// TIA Portal project "cpsforge_tiaportal" (V17)

(* hardware
DEVICE "S7-1200 station_1"  S7-1200 Station
   slot 0: "Rack_0"  S7-1200 Rack  Rack  V1.0
   slot 1: "PLC_1"  CPU 1212FC DC/DC/RLY  6ES7 212-1HF40-0XB0  V4.5
*)

// ===== PLC "PLC_1"  CPU 1212FC DC/DC/RLY =====

VAR_GLOBAL   // PLC tag table "Default tag table"
   "Tag__639094376035440745" AT %I0.0 : Bool;
   "Tag__639094376037924724" AT %Q0.0 : Bool;
   "Tag__639094376037924725" AT %I0.1 : Bool;
   "Tag__639094376038085904" AT %Q0.1 : Bool;
   "Tag__639094376038085905" AT %Q0.2 : Bool;
   "Tag__639094376038245632" AT %I0.2 : Bool;
   "Tag__639094376038245633" AT %I0.3 : Bool;
   "Tag__639094376038405651" AT %I0.4 : Bool;
   "Tag__639094376038405652" AT %I0.5 : Bool;
   "Tag__639094376038405653" AT %Q0.3 : Bool;
   "Tag__639094376038565707" AT %Q0.4 : Bool;
   "Tag__639094376038565708" AT %Q0.5 : Bool;
   "Tag__639094376038565709" AT %Q1.0 : Bool;
   "Tag__639094376038885860" AT %I10.0 : Bool;
   "Tag__639094376038885861" AT %I10.1 : Bool;
   "Tag__639094376039046363" AT %I10.2 : Bool;
   "Tag__639094376039046364" AT %I10.3 : Bool;
   "Tag__639094376039046365" AT %I10.4 : Bool;
   "Tag__639094376039205258" AT %I10.5 : Bool;
   "Tag__639094376039205259" AT %I10.6 : Bool;
   "Tag__639094376039205260" AT %I10.7 : Bool;
   "Tag__639094376039365268" AT %I11.0 : Bool;
   "Tag__639094376039365269" AT %I11.1 : Bool;
   "Tag__639094376039365270" AT %I11.2 : Bool;
   "Tag__639094376039525211" AT %I11.3 : Bool;
   "Tag__639094376039525212" AT %I11.4 : Bool;
   "Tag__639094376039525213" AT %I11.5 : Bool;
   "Tag__639094376039685481" AT %I11.6 : Bool;
   "Tag__639094376039685482" AT %I11.7 : Bool;
   "Tag__639094376039685483" AT %I12.0 : Bool;
   "Tag__639094376039846408" AT %I12.1 : Bool;
   "Tag__639094376039846409" AT %I12.2 : Bool;
   "Tag__639094376039846410" AT %Q0.6 : Bool;
   "Tag__639094376040005546" AT %Q0.7 : Bool;
   "Tag__639094376040005547" AT %Q1.1 : Bool;
   "Tag__639094376040005548" AT %Q1.2 : Bool;
   "Tag__639094376040163908" AT %Q1.3 : Bool;
   "Tag__639094376040163909" AT %Q1.4 : Bool;
   "Tag__639094376040163910" AT %Q1.5 : Bool;
   "Tag__639094376040323143" AT %Q1.6 : Bool;
   "Tag__639094376040323144" AT %Q1.7 : Bool;
   "Tag__639094376040323145" AT %Q2.0 : Bool;
   "Tag__639094376040483081" AT %Q2.1 : Bool;
   "Tag__639094376040483082" AT %Q2.2 : Bool;
   "Tag__639094376040483083" AT %Q2.3 : Bool;
   "Tag__639094376040642647" AT %Q2.4 : Bool;
   "Tag__639094376040642648" AT %Q2.5 : Bool;
   "Tag__639094376040642649" AT %Q2.6 : Bool;
   "Tag__639094376040802767" AT %Q2.7 : Bool;
   "Tag__639094376040802768" AT %Q3.0 : Bool;
   "Tag__639094376040802769" AT %Q3.1 : Bool;
   "Tag__639094376040963045" AT %QD100 : DWord;
   "Tag__639094376041124518" AT %I12.3 : Bool;
   "Tag__639094376041124519" AT %I12.4 : Bool;
   "Tag__639094376041283188" AT %I12.5 : Bool;
   "Tag__639094376041283189" AT %I12.6 : Bool;
   "Tag__639094376041283190" AT %I12.7 : Bool;
   "Tag__639094376041442043" AT %I13.0 : Bool;
   "Tag__639094376041442044" AT %I13.1 : Bool;
   "Tag__639094376041600752" AT %I13.2 : Bool;
   "Tag__639094376041600753" AT %I13.3 : Bool;
   "Tag__639094376041600754" AT %I13.4 : Bool;
   "Tag__639094376041760860" AT %Q3.2 : Bool;
   "Tag__639094376041918319" AT %Q3.3 : Bool;
   "Tag__639094376041918320" AT %Q3.4 : Bool;
   "Tag__639094376042076147" AT %ID100 : DWord;
   "Tag__639094376042076148" AT %ID104 : DWord;
   "Tag__639094376042235578" AT %ID108 : DWord;
   "Tag__639094376042315926" AT %QD104 : DWord;
   "Tag__639094376042397245" AT %QD108 : DWord;
   "Tag__639094376042397246" AT %QD112 : DWord;
   "Tag__639094376042713202" AT %I0.6 : Bool;
   "Tag__639094376042871627" AT %I0.7 : Bool;
   "Tag__639094376042871628" AT %I1.0 : Bool;
   "Tag__639094376043030339" AT %I1.1 : Bool;
   "Tag__639094376043070322" AT %I1.2 : Bool;
   "Tag__639094376043147186" AT %I1.3 : Bool;
   "Tag__639094376043188096" AT %I1.4 : Bool;
   "Tag__639094376043188097" AT %I1.5 : Bool;
   "Tag__639094376043188098" AT %I1.6 : Bool;
   "Tag__639094376043345950" AT %I1.7 : Bool;
   "Tag__639094559022291825" AT %QB0 : Byte;
   "Tag__639094559022387271" AT %QB1 : Byte;
   "Tag__639094559022442425" AT %QB2 : Byte;
   "Tag__639094559022502581" AT %QB3 : Byte;
END_VAR

DATA_BLOCK "DB_Config"   // DB2
{ S7_Optimized_Access := 'FALSE' }
VERSION : 0.1
// MANTIS â€” DB_Config: Global configuration block
//  ActiveScene selects which Factory I/O scene is running
   VAR
      ActiveScene : Int := 19;   // Default: Sorting Height Basic
      ScanRate_ms : Int := 1000;   // Control loop period
      Running : Bool := TRUE;   // System running flag
   END_VAR
BEGIN
END_DATA_BLOCK

DATA_BLOCK "FB_FromAtoB_DB"   // DB3
{ S7_Optimized_Access := 'FALSE' }
VERSION : 0.1
// =============================================================================
//  MANTIS â€” Instance Data Blocks for all 21 Factory I/O Scene FBs
// 
//  After importing this file in TIA Portal, you MUST set the DB numbers:
//    Right-click each DB â†’ Properties â†’ General â†’ Number
//    Assign the DB numbers according to the table below.
// 
//  DB Number Assignments:
//    DB10 = FB_FromAtoB_DB
//    DB11 = FB_FromAtoB_SR_DB
//    DB12 = FB_FillingTank_DB
//    DB13 = FB_QueueItems_DB
//    DB14 = FB_Assembler_DB
//    DB15 = FB_AssemblerAnalog_DB
//    DB16 = FB_Warehouse_DB
//    DB17 = FB_BufferStation_DB
//    DB18 = FB_ConvergeStation_DB
//    DB19 = FB_ElevatorAdvanced_DB
//    DB20 = FB_ElevatorBasic_DB
//    DB21 = FB_LevelControl_DB
//    DB22 = FB_Palletizer_DB
//    DB23 = FB_PickPlaceBasic_DB
//    DB24 = FB_PickPlaceXYZ_DB
//    DB25 = FB_ProductionLine_DB
//    DB26 = FB_SeparatingStation_DB
//    DB27 = FB_SortingHeightAdv_DB
//    DB28 = FB_SortingHeightBasic_DB
//    DB29 = FB_SortingWeight_DB
//    DB30 = FB_SortingStation_DB
//  =============================================================================
//  Scene 1: From A to B â†’ DB10
// stored: InstanceOfName FB_FromAtoB
"FB_FromAtoB"
BEGIN
END_DATA_BLOCK

DATA_BLOCK "FB_FromAtoB_SR_DB"   // DB4
{ S7_Optimized_Access := 'FALSE' }
VERSION : 0.1
// Scene 2: From A to B (Set/Reset) â†’ DB11
// stored: InstanceOfName FB_FromAtoB_SR
"FB_FromAtoB_SR"
BEGIN
END_DATA_BLOCK

DATA_BLOCK "FB_FillingTank_DB"   // DB5
{ S7_Optimized_Access := 'FALSE' }
VERSION : 0.1
// Scene 3: Filling Tank â†’ DB12
// stored: InstanceOfName FB_FillingTank
"FB_FillingTank"
BEGIN
END_DATA_BLOCK

DATA_BLOCK "FB_QueueItems_DB"   // DB6
{ S7_Optimized_Access := 'FALSE' }
VERSION : 0.1
// Scene 4: Queue of Items â†’ DB13
// stored: InstanceOfName FB_QueueItems
"FB_QueueItems"
BEGIN
END_DATA_BLOCK

DATA_BLOCK "FB_Assembler_DB"   // DB7
{ S7_Optimized_Access := 'FALSE' }
VERSION : 0.1
// Scene 5: Assembler â†’ DB14
// stored: InstanceOfName FB_Assembler
"FB_Assembler"
BEGIN
END_DATA_BLOCK

DATA_BLOCK "FB_AssemblerAnalog_DB"   // DB8
{ S7_Optimized_Access := 'FALSE' }
VERSION : 0.1
// Scene 6: Assembler (Analog) â†’ DB15
// stored: InstanceOfName FB_AssemblerAnalog
"FB_AssemblerAnalog"
BEGIN
END_DATA_BLOCK

DATA_BLOCK "FB_Warehouse_DB"   // DB9
{ S7_Optimized_Access := 'FALSE' }
VERSION : 0.1
// Scene 7: Automated Warehouse â†’ DB16
// stored: InstanceOfName FB_Warehouse
"FB_Warehouse"
BEGIN
END_DATA_BLOCK

DATA_BLOCK "FB_BufferStation_DB"   // DB10
{ S7_Optimized_Access := 'FALSE' }
VERSION : 0.1
// Scene 8: Buffer Station â†’ DB17
// stored: InstanceOfName FB_BufferStation
"FB_BufferStation"
BEGIN
END_DATA_BLOCK

DATA_BLOCK "FB_ConvergeStation_DB"   // DB11
{ S7_Optimized_Access := 'FALSE' }
VERSION : 0.1
// Scene 9: Converge Station â†’ DB18
// stored: InstanceOfName FB_ConvergeStation
"FB_ConvergeStation"
BEGIN
END_DATA_BLOCK

DATA_BLOCK "FB_ElevatorAdvanced_DB"   // DB12
{ S7_Optimized_Access := 'FALSE' }
VERSION : 0.1
// Scene 10: Elevator (Advanced) â†’ DB19
// stored: InstanceOfName FB_ElevatorAdvanced
"FB_ElevatorAdvanced"
BEGIN
END_DATA_BLOCK

DATA_BLOCK "FB_ElevatorBasic_DB"   // DB13
{ S7_Optimized_Access := 'FALSE' }
VERSION : 0.1
// Scene 11: Elevator (Basic) â†’ DB20
// stored: InstanceOfName FB_ElevatorBasic
"FB_ElevatorBasic"
BEGIN
END_DATA_BLOCK

DATA_BLOCK "FB_LevelControl_DB"   // DB14
{ S7_Optimized_Access := 'FALSE' }
VERSION : 0.1
// Scene 12: Level Control â†’ DB21
// stored: InstanceOfName FB_LevelControl
"FB_LevelControl"
BEGIN
END_DATA_BLOCK

DATA_BLOCK "FB_Palletizer_DB"   // DB15
{ S7_Optimized_Access := 'FALSE' }
VERSION : 0.1
// Scene 13: Palletizer â†’ DB22
// stored: InstanceOfName FB_Palletizer
"FB_Palletizer"
BEGIN
END_DATA_BLOCK

DATA_BLOCK "FB_PickPlaceBasic_DB"   // DB16
{ S7_Optimized_Access := 'FALSE' }
VERSION : 0.1
// Scene 14: Pick & Place (Basic) â†’ DB23
// stored: InstanceOfName FB_PickPlaceBasic
"FB_PickPlaceBasic"
BEGIN
END_DATA_BLOCK

DATA_BLOCK "FB_PickPlaceXYZ_DB"   // DB17
{ S7_Optimized_Access := 'FALSE' }
VERSION : 0.1
// Scene 15: Pick & Place XYZ â†’ DB24
// stored: InstanceOfName FB_PickPlaceXYZ
"FB_PickPlaceXYZ"
BEGIN
END_DATA_BLOCK

DATA_BLOCK "FB_ProductionLine_DB"   // DB18
{ S7_Optimized_Access := 'FALSE' }
VERSION : 0.1
// Scene 16: Production Line â†’ DB25
// stored: InstanceOfName FB_ProductionLine
"FB_ProductionLine"
BEGIN
END_DATA_BLOCK

DATA_BLOCK "FB_SeparatingStation_DB"   // DB19
{ S7_Optimized_Access := 'FALSE' }
VERSION : 0.1
// Scene 17: Separating Station â†’ DB26
// stored: InstanceOfName FB_SeparatingStation
"FB_SeparatingStation"
BEGIN
END_DATA_BLOCK

DATA_BLOCK "FB_SortingHeightAdv_DB"   // DB20
{ S7_Optimized_Access := 'FALSE' }
VERSION : 0.1
// Scene 18: Sorting by Height (Advanced) â†’ DB27
// stored: InstanceOfName FB_SortingHeightAdvanced
"FB_SortingHeightAdvanced"
BEGIN
END_DATA_BLOCK

DATA_BLOCK "FB_SortingHeightBasic_DB"   // DB21
{ S7_Optimized_Access := 'FALSE' }
VERSION : 0.1
// Scene 19: Sorting by Height (Basic) â†’ DB28
// stored: InstanceOfName FB_SortingHeightBasic
"FB_SortingHeightBasic"
BEGIN
END_DATA_BLOCK

DATA_BLOCK "FB_SortingWeight_DB"   // DB22
{ S7_Optimized_Access := 'FALSE' }
VERSION : 0.1
// Scene 20: Sorting by Weight â†’ DB29
// stored: InstanceOfName FB_SortingWeight
"FB_SortingWeight"
BEGIN
END_DATA_BLOCK

DATA_BLOCK "FB_SortingStation_DB"   // DB23
{ S7_Optimized_Access := 'FALSE' }
VERSION : 0.1
// Scene 21: Sorting Station â†’ DB30
// stored: InstanceOfName FB_SortingStation
"FB_SortingStation"
BEGIN
END_DATA_BLOCK

FUNCTION_BLOCK "FB_Assembler"   // FB2, SCL
{ S7_Optimized_Access := 'FALSE' }
VERSION : 0.1
// MANTIS â€” Scene 5: Assembler
//  Assemble parts (lids + bases) using a two-axis pick and place.
//  DB14: I/O mapping
   VAR
      PartAtPickup : Bool;   // 0.0
      _pad0 : Byte;
      PartAtPlace : Bool;   // 2.0
      _pad1 : Byte;
      LidAtPickup : Bool;   // 4.0
      _pad2 : Byte;
      ClampSensor : Bool;   // 6.0
      _pad3 : Byte;
      MovingX : Bool;   // 8.0
      _pad4 : Byte;
      MovingZ : Bool;   // 10.0
      _pad5 : Byte;
      ConveyorBase : Bool;   // 12.0
      _pad6 : Byte;
      ConveyorLid : Bool;   // 14.0
      _pad7 : Byte;
      ConveyorOut : Bool;   // 16.0
      _pad8 : Byte;
      MoveX : Bool;   // 18.0
      _pad9 : Byte;
      MoveZ : Bool;   // 20.0
      _pad10 : Byte;
      Clamp : Bool;   // 22.0
      _pad11 : Byte;
      Emitter : Bool;   // 24.0
      _pad12 : Byte;
      iState : Int := 0;
   END_VAR
BEGIN
       CASE #iState OF
           0: // Feed base part
               #ConveyorBase := TRUE;
               #ConveyorLid := TRUE;
               #Emitter := TRUE;
               IF #PartAtPickup THEN
                   #ConveyorBase := FALSE;
                   #iState := 1;
               END_IF;

           1: // Move pick-and-place to pickup position
               #MoveX := FALSE;  // Move to pickup (left)
               #MoveZ := TRUE;   // Lower
               IF NOT #MovingZ THEN
                   #iState := 2;
               END_IF;

           2: // Clamp the part
               #Clamp := TRUE;
               IF #ClampSensor THEN
                   #MoveZ := FALSE;  // Raise
                   #iState := 3;
               END_IF;

           3: // Move to place position
               IF NOT #MovingZ THEN
                   #MoveX := TRUE;   // Move to place (right)
                   #iState := 4;
               END_IF;

           4: // Lower and place
               IF NOT #MovingX THEN
                   #MoveZ := TRUE;   // Lower
                   #iState := 5;
               END_IF;

           5: // Release
               IF NOT #MovingZ THEN
                   #Clamp := FALSE;
                   #MoveZ := FALSE;
                   #iState := 6;
               END_IF;

           6: // Output assembled part
               #ConveyorOut := TRUE;
               #MoveX := FALSE;  // Return to home
               IF NOT #PartAtPlace THEN
                   #ConveyorOut := FALSE;
                   #iState := 0;
               END_IF;
       END_CASE;
END_FUNCTION_BLOCK

FUNCTION_BLOCK "FB_AssemblerAnalog"   // FB3, SCL
{ S7_Optimized_Access := 'FALSE' }
VERSION : 0.1
// MANTIS â€” Scene 6: Assembler (Analog)
//  Assemble with analog position control for X/Z axes.
//  DB15: I/O mapping
   VAR
      PartAtPickup : Bool;   // 0.0
      _pad0 : Byte;
      PartAtPlace : Bool;   // 2.0
      _pad1 : Byte;
      LidAtPickup : Bool;   // 4.0
      _pad2 : Byte;
      ClampSensor : Bool;   // 6.0
      _pad3 : Byte;
      PosX : Real;   // 8
      PosZ : Real;   // 12
      ConveyorBase : Bool;   // 16.0
      _pad4 : Byte;
      ConveyorLid : Bool;   // 18.0
      _pad5 : Byte;
      ConveyorOut : Bool;   // 20.0
      _pad6 : Byte;
      SetpointX : Real;   // 22
      SetpointZ : Real;   // 26
      Clamp : Bool;   // 30.0
      _pad7 : Byte;
      Emitter : Bool;   // 32.0
      _pad8 : Byte;
      iState : Int := 0;
      PICKUP_X : Real := 100.0;
      PICKUP_Z : Real := 400.0;
      PLACE_X : Real := 800.0;
      PLACE_Z : Real := 400.0;
      HOME_Z : Real := 50.0;
      TOLERANCE : Real := 10.0;
   END_VAR
BEGIN
       CASE #iState OF
           0: // Feed parts
               #ConveyorBase := TRUE;
               #ConveyorLid := TRUE;
               #Emitter := TRUE;
               #SetpointX := #PICKUP_X;
               #SetpointZ := #HOME_Z;
               IF #PartAtPickup THEN
                   #ConveyorBase := FALSE;
                   #iState := 1;
               END_IF;

           1: // Move to pickup and lower
               #SetpointX := #PICKUP_X;
               #SetpointZ := #PICKUP_Z;
               IF ABS(#PosX - #PICKUP_X) < #TOLERANCE AND ABS(#PosZ - #PICKUP_Z) < #TOLERANCE THEN
                   #iState := 2;
               END_IF;

           2: // Clamp
               #Clamp := TRUE;
               IF #ClampSensor THEN
                   #SetpointZ := #HOME_Z;
                   #iState := 3;
               END_IF;

           3: // Raise and move to place
               IF ABS(#PosZ - #HOME_Z) < #TOLERANCE THEN
                   #SetpointX := #PLACE_X;
                   #iState := 4;
               END_IF;

           4: // Lower to place
               IF ABS(#PosX - #PLACE_X) < #TOLERANCE THEN
                   #SetpointZ := #PLACE_Z;
                   #iState := 5;
               END_IF;

           5: // Release
               IF ABS(#PosZ - #PLACE_Z) < #TOLERANCE THEN
                   #Clamp := FALSE;
                   #SetpointZ := #HOME_Z;
                   #iState := 6;
               END_IF;

           6: // Output
               #ConveyorOut := TRUE;
               #SetpointX := #PICKUP_X;
               IF NOT #PartAtPlace THEN
                   #ConveyorOut := FALSE;
                   #iState := 0;
               END_IF;
       END_CASE;
END_FUNCTION_BLOCK

FUNCTION_BLOCK "FB_BufferStation"   // FB4, SCL
{ S7_Optimized_Access := 'FALSE' }
VERSION : 0.2
// MANTIS â€” Scene 8: Buffer Station
//  Buffer and separate up to five boxes.
//  DB17: I/O mapping
   VAR
      Sensor1 : Bool;   // 0.0
      _pad0 : Byte;
      Sensor2 : Bool;   // 2.0
      _pad1 : Byte;
      Sensor3 : Bool;   // 4.0
      _pad2 : Byte;
      Sensor4 : Bool;   // 6.0
      _pad3 : Byte;
      Sensor5 : Bool;   // 8.0
      _pad4 : Byte;
      AtExit : Bool;   // 10.0
      _pad5 : Byte;
      Conveyor : Bool;   // 12.0
      _pad6 : Byte;
      Stopper1 : Bool;   // 14.0
      _pad7 : Byte;
      Stopper2 : Bool;   // 16.0
      _pad8 : Byte;
      Emitter : Bool;   // 18.0
      _pad9 : Byte;
      Remover : Bool;   // 20.0
      _pad10 : Byte;
      iState : Int := 0;
      BoxCount : Int := 0;
      BUFFER_MAX : Int := 5;
   END_VAR
BEGIN
       // Always-on infrastructure
       #Conveyor := TRUE;
       #Emitter := TRUE;
       #Remover := TRUE;

       // Count boxes by number of occupied sensor positions
       #BoxCount := 0;
       IF #Sensor1 THEN
           #BoxCount := #BoxCount + 1;
       END_IF;
       IF #Sensor2 THEN
           #BoxCount := #BoxCount + 1;
       END_IF;
       IF #Sensor3 THEN
           #BoxCount := #BoxCount + 1;
       END_IF;
       IF #Sensor4 THEN
           #BoxCount := #BoxCount + 1;
       END_IF;
       IF #Sensor5 THEN
           #BoxCount := #BoxCount + 1;
       END_IF;

       // Simple pass-through with stoppers open
       // Stopper FALSE = retracted (passing), TRUE = extended (blocking)
       // Let boxes flow freely â€” Remover handles cleanup at exit
       CASE #iState OF
           0: // Accumulate: both stoppers open, let boxes fill buffer
               #Stopper1 := FALSE;
               #Stopper2 := FALSE;
               IF #BoxCount >= #BUFFER_MAX THEN
                   // Buffer full â€” close entry stopper to stop more
                   #Stopper1 := TRUE;
                   #iState := 1;
               END_IF;

           1: // Buffer full â€” hold and release one at a time
               #Stopper1 := TRUE;   // Block new arrivals
               #Stopper2 := FALSE;  // Let exit box through
               IF #AtExit THEN
                   #iState := 2;
               END_IF;

           2: // Wait for exit to clear, then go back to accumulate
               #Stopper1 := TRUE;
               #Stopper2 := FALSE;
               IF NOT #AtExit THEN
                   #iState := 0;
               END_IF;
       END_CASE;
END_FUNCTION_BLOCK

FUNCTION_BLOCK "FB_ConvergeStation"   // FB5, SCL
{ S7_Optimized_Access := 'FALSE' }
VERSION : 0.2
// MANTIS â€” Scene 9: Converge Station
//  Converge two paths into a single output conveyor.
//  DB18: I/O mapping
   VAR
      SensorLeft : Bool;   // 0.0
      _pad0 : Byte;
      SensorRight : Bool;   // 2.0
      _pad1 : Byte;
      SensorMerge : Bool;   // 4.0
      _pad2 : Byte;
      AtExit : Bool;   // 6.0
      _pad3 : Byte;
      ConveyorLeft : Bool;   // 8.0
      _pad4 : Byte;
      ConveyorRight : Bool;   // 10.0
      _pad5 : Byte;
      ConveyorOut : Bool;   // 12.0
      _pad6 : Byte;
      Emitter1 : Bool;   // 14.0
      _pad7 : Byte;
      Emitter2 : Bool;   // 16.0
      _pad8 : Byte;
      Remover : Bool;   // 18.0
      _pad9 : Byte;
      Priority : Bool := FALSE;   // FALSE=left first, TRUE=right first
   END_VAR
BEGIN
       // Always-on infrastructure
       #ConveyorOut := TRUE;
       #Remover := TRUE;
       #Emitter1 := TRUE;
       #Emitter2 := TRUE;

       // Default: run BOTH input conveyors so boxes reach sensors
       #ConveyorLeft := TRUE;
       #ConveyorRight := TRUE;

       IF #SensorMerge THEN
           // Merge point occupied â€” stop both inputs, toggle priority for next
           #ConveyorLeft := FALSE;
           #ConveyorRight := FALSE;
           #Priority := NOT #Priority;
       ELSIF #SensorLeft AND #SensorRight THEN
           // Both sides have a box â€” let priority side through, hold the other
           IF #Priority THEN
               #ConveyorLeft := FALSE;   // Hold left, let right advance
           ELSE
               #ConveyorRight := FALSE;  // Hold right, let left advance
           END_IF;
       END_IF;
       // If only one side has a box, both conveyors stay on â†’ box advances freely
END_FUNCTION_BLOCK

FUNCTION_BLOCK "FB_ElevatorAdvanced"   // FB6, SCL
{ S7_Optimized_Access := 'FALSE' }
VERSION : 0.4
// MANTIS â€” Scene 10: Elevator (Advanced)
//  Single elevator servicing 4 floors (0-3), collecting items into a box.
//  DB19: Instance DB (non-optimized access)
// 
//  OBJECTIVE: Collect exactly 5 items into a stackable box using the elevator.
//    Items arrive randomly at floors 1-3. The elevator carries a box, visits
//    each floor with waiting items, loads items into the box, and after 5 items
//    are collected, returns to floor 0 to unload the full box. A new empty box
//    is then loaded and the cycle repeats.
// 
//  Factory I/O layout:
//    4-floor structure with a single elevator shaft.
//    Items spawn randomly at floors 1-3 (emitters on auto).
//    Box sits on elevator platform, items loaded into box at each floor.
//    After 5 items collected, box exits at floor 0 (remover on auto).
//    Control panel with Start/Stop/Reset/EmergencyStop/Auto.
//    Traffic lights per floor (Green/Yellow/Red for floors 1-3).
//    Floor indicator lights (Floor 1/2/3).
//    Display shows items collected (ItemCount).
// 
//  Driver mapping (from Factory I/O):
//    SENSORS (Inputs): NOTE â€” remapped to %I10.x+ to avoid S7-1200 built-in DI conflict
//      At 1             â†’ %I10.0  (floor 1 call)
//      At 2             â†’ %I10.1  (floor 2 call)
//      At 3             â†’ %I10.2  (floor 3 call)
//      At elevator      â†’ %I10.3  (item on elevator)
//      At entry         â†’ %I10.4  (item at entry)
//      At exit          â†’ %I10.5  (item at exit)
//      At 0 (low)       â†’ %I10.6
//      At 0 (high)      â†’ %I10.7
//      At 1 (low)       â†’ %I11.0
//      At 1 (high)      â†’ %I11.1
//      At 2 (low)       â†’ %I11.2
//      At 2 (high)      â†’ %I11.3
//      At 3 (low)       â†’ %I11.4
//      At 3 (high)      â†’ %I11.5
//      Start            â†’ %I11.6
//      Reset            â†’ %I11.7
//      Stop             â†’ %I12.0
//      Emergency stop   â†’ %I12.1
//      Auto             â†’ %I12.2
//      FACTORY I/O (Running) â†’ %I12.3
// 
//    ACTUATORS (Outputs):
//      Conveyor 0       â†’ %Q0.0
//      Conveyor 1       â†’ %Q0.1
//      Conveyor 2       â†’ %Q0.2
//      Conveyor 3       â†’ %Q0.3
//      Exit conveyor    â†’ %Q0.4
//      Load             â†’ %Q0.5
//      Unload           â†’ %Q0.6
//      Up               â†’ %Q0.7
//      Down             â†’ %Q1.0
//      Slow             â†’ %Q1.1
//      Warning light    â†’ %Q1.2
//      Start light      â†’ %Q1.3
//      Reset light      â†’ %Q1.4
//      Stop light       â†’ %Q1.5
//      Floor 1          â†’ %Q1.6
//      Floor 2          â†’ %Q1.7
//      Floor 3          â†’ %Q2.0
//      Green 1          â†’ %Q2.1
//      Yellow 1         â†’ %Q2.2
//      Red 1            â†’ %Q2.3
//      Green 2          â†’ %Q2.4
//      Yellow 2         â†’ %Q2.5
//      Red 2            â†’ %Q2.6
//      Green 3          â†’ %Q2.7
//      Yellow 3         â†’ %Q3.0
//      Red 3            â†’ %Q3.1
//      Display          â†’ (DINT) %QD100
// 
//  DB19 byte layout (non-optimized):
//    Sensors:
//      0:  At1          2: At2          4: At3
//      6:  AtElevator   8: AtEntry     10: AtExit
//     12:  At0Low      14: At0High     16: At1Low
//     18:  At1High     20: At2Low      22: At2High
//     24:  At3Low      26: At3High
//     28:  BtnStart    30: BtnReset    32: BtnStop
//     34:  EmergencyStop  36: BtnAuto
//    Actuators:
//     38:  Conveyor0   40: Conveyor1   42: Conveyor2
//     44:  Conveyor3   46: ExitConveyor
//     48:  Load        50: Unload
//     52:  Up          54: Down        56: Slow
//     58:  WarningLight
//     60:  StartLight  62: ResetLight  64: StopLight
//     66:  Floor1Ind   68: Floor2Ind   70: Floor3Ind
//     72:  Green1      74: Yellow1     76: Red1
//     78:  Green2      80: Yellow2     82: Red2
//     84:  Green3      86: Yellow3     88: Red3
//     90-93: Display (DINT)
//    Internal:
//     94:  iState (INT)      96: TargetFloor (INT)
//     98:  CurrentFloor (INT) 100: DwellTimer (INT)
//    102:  Running (BOOL)   104: Enable (BOOL)
//    106:  ItemCount (INT)  108: MaxItems (INT, default 5)
//    Total = 110 bytes
// 
//  State machine (6 states):
//    S0 = LOAD_BOX:  At floor 0, load new empty box onto elevator
//    S1 = SCAN:      Check floors 1-3 for waiting items
//    S2 = MOVING:    Go to target floor
//    S3 = COLLECT:   At target floor, load item into box, increment ItemCount
//    S4 = RETURN:    Box full (ItemCount >= MaxItems), go back to floor 0
//    S5 = UNLOAD:    At floor 0, push full box off, reset ItemCount
// 
//  Vulnerability: Enable (byte 104) â€” read but NEVER written by PLC.
//  Attack vectors:
//    - ItemCount (byte 106): set to 5 early â†’ box exits with fewer items
//    - ItemCount (byte 106): reset to 0 â†’ box never exits, items overflow
//    - MaxItems (byte 108): set to 1 â†’ box exits after 1 item
//    - Enable (byte 104): set FALSE â†’ system shuts down completely
//  â”€â”€ Sensors (inputs) â”€â”€
   VAR
      At1 : Bool;   // byte 0 â€” %I10.0 floor 1 call
      _p00 : Byte;
      At2 : Bool;   // byte 2 â€” %I10.1 floor 2 call
      _p01 : Byte;
      At3 : Bool;   // byte 4 â€” %I10.2 floor 3 call
      _p02 : Byte;
      AtElevator : Bool;   // byte 6 â€” %I10.3 item on elevator
      _p03 : Byte;
      AtEntry : Bool;   // byte 8 â€” %I10.4 item at entry
      _p04 : Byte;
      AtExit : Bool;   // byte 10 â€” %I10.5 item at exit
      _p05 : Byte;
      At0Low : Bool;   // byte 12 â€” %I10.6 elevator near floor 0
      _p06 : Byte;
      At0High : Bool;   // byte 14 â€” %I10.7 elevator at floor 0
      _p07 : Byte;
      At1Low : Bool;   // byte 16 â€” %I11.0 elevator near floor 1
      _p08 : Byte;
      At1High : Bool;   // byte 18 â€” %I11.1 elevator at floor 1
      _p09 : Byte;
      At2Low : Bool;   // byte 20 â€” %I11.2 elevator near floor 2
      _p10 : Byte;
      At2High : Bool;   // byte 22 â€” %I11.3 elevator at floor 2
      _p11 : Byte;
      At3Low : Bool;   // byte 24 â€” %I11.4 elevator near floor 3
      _p12 : Byte;
      At3High : Bool;   // byte 26 â€” %I11.5 elevator at floor 3
      _p13 : Byte;
      BtnStart : Bool;   // byte 28 â€” %I11.6
      _p14 : Byte;
      BtnReset : Bool;   // byte 30 â€” %I11.7
      _p15 : Byte;
      BtnStop : Bool;   // byte 32 â€” %I12.0
      _p16 : Byte;
      EmergencyStop : Bool;   // byte 34 â€” %I12.1
      _p17 : Byte;
      BtnAuto : Bool;   // byte 36 â€” %I12.2
      _p18 : Byte;   // â”€â”€ Actuators (outputs) â”€â”€
      Conveyor0 : Bool;   // byte 38 â€” %Q0.0
      _p19 : Byte;
      Conveyor1 : Bool;   // byte 40 â€” %Q0.1
      _p20 : Byte;
      Conveyor2 : Bool;   // byte 42 â€” %Q0.2
      _p21 : Byte;
      Conveyor3 : Bool;   // byte 44 â€” %Q0.3
      _p22 : Byte;
      ExitConveyor : Bool;   // byte 46 â€” %Q0.4
      _p23 : Byte;
      Load : Bool;   // byte 48 â€” %Q0.5
      _p24 : Byte;
      Unload : Bool;   // byte 50 â€” %Q0.6
      _p25 : Byte;
      Up : Bool;   // byte 52 â€” %Q0.7
      _p26 : Byte;
      Down : Bool;   // byte 54 â€” %Q1.0
      _p27 : Byte;
      Slow : Bool;   // byte 56 â€” %Q1.1
      _p28 : Byte;
      WarningLight : Bool;   // byte 58 â€” %Q1.2
      _p29 : Byte;
      StartLight : Bool;   // byte 60 â€” %Q1.3
      _p30 : Byte;
      ResetLight : Bool;   // byte 62 â€” %Q1.4
      _p31 : Byte;
      StopLight : Bool;   // byte 64 â€” %Q1.5
      _p32 : Byte;
      Floor1Ind : Bool;   // byte 66 â€” %Q1.6
      _p33 : Byte;
      Floor2Ind : Bool;   // byte 68 â€” %Q1.7
      _p34 : Byte;
      Floor3Ind : Bool;   // byte 70 â€” %Q2.0
      _p35 : Byte;
      Green1 : Bool;   // byte 72 â€” %Q2.1
      _p36 : Byte;
      Yellow1 : Bool;   // byte 74 â€” %Q2.2
      _p37 : Byte;
      Red1 : Bool;   // byte 76 â€” %Q2.3
      _p38 : Byte;
      Green2 : Bool;   // byte 78 â€” %Q2.4
      _p39 : Byte;
      Yellow2 : Bool;   // byte 80 â€” %Q2.5
      _p40 : Byte;
      Red2 : Bool;   // byte 82 â€” %Q2.6
      _p41 : Byte;
      Green3 : Bool;   // byte 84 â€” %Q2.7
      _p42 : Byte;
      Yellow3 : Bool;   // byte 86 â€” %Q3.0
      _p43 : Byte;
      Red3 : Bool;   // byte 88 â€” %Q3.1
      _p44 : Byte;
      Display : DInt;   // byte 90 â€” %QD100 (floor display) â”€â”€ Internal state â”€â”€
      iState : Int := 0;   // byte 94 â€” state machine
      TargetFloor : Int := 0;   // byte 96 â€” where to go (0-3)
      CurrentFloor : Int := 0;   // byte 98 â€” last known floor
      DwellTimer : Int := 0;   // byte 100 â€” load/unload dwell
      Running : Bool := FALSE;   // byte 102 â€” system running
      _p45 : Byte;
      Enable : Bool := TRUE;   // byte 104 â€” system enable (default ON)
      _p46 : Byte;
      ItemCount : Int := 0;   // byte 106 â€” items collected in current box
      MaxItems : Int := 5;   // byte 108 â€” target items per box (default 5) Total: 110 bytes
   END_VAR
   VAR_TEMP
      atTarget : Bool;
      nearTarget : Bool;
   END_VAR
BEGIN
       // â•â•â•â•â•â•â•â•â•â•â•â•â•â•â•â•â•â•â•â•â•â•â•â•â•â•â•â•â•â•â•â•â•â•â•â•â•â•â•â•â•â•â•â•â•â•â•â•â•â•â•â•
       // Safety gate: if Enable is FALSE, shut everything down
       // â•â•â•â•â•â•â•â•â•â•â•â•â•â•â•â•â•â•â•â•â•â•â•â•â•â•â•â•â•â•â•â•â•â•â•â•â•â•â•â•â•â•â•â•â•â•â•â•â•â•â•â•
       IF NOT #Enable THEN
           #Running := FALSE;
           #Up := FALSE;
           #Down := FALSE;
           #Slow := FALSE;
           #Load := FALSE;
           #Unload := FALSE;
           #Conveyor0 := FALSE;
           #Conveyor1 := FALSE;
           #Conveyor2 := FALSE;
           #Conveyor3 := FALSE;
           #ExitConveyor := FALSE;
           #WarningLight := TRUE;
           #StartLight := FALSE;
           #StopLight := TRUE;
           #ResetLight := FALSE;
           #Floor1Ind := FALSE;
           #Floor2Ind := FALSE;
           #Floor3Ind := FALSE;
           #Green1 := FALSE;
           #Yellow1 := FALSE;
           #Red1 := TRUE;
           #Green2 := FALSE;
           #Yellow2 := FALSE;
           #Red2 := TRUE;
           #Green3 := FALSE;
           #Yellow3 := FALSE;
           #Red3 := TRUE;
           #Display := 0;
           RETURN;
       END_IF;

       // â•â•â•â•â•â•â•â•â•â•â•â•â•â•â•â•â•â•â•â•â•â•â•â•â•â•â•â•â•â•â•â•â•â•â•â•â•â•â•â•â•â•â•â•â•â•â•â•â•â•â•â•
       // Button handling (NC buttons: TRUE = safe/not pressed)
       //   EmergencyStop: TRUE = not activated (safe)
       //   BtnStop: TRUE = not pressed (safe)
       //   BtnStart: TRUE = pressed (momentary)
       // Auto-start: when safe conditions met and system not running
       // â•â•â•â•â•â•â•â•â•â•â•â•â•â•â•â•â•â•â•â•â•â•â•â•â•â•â•â•â•â•â•â•â•â•â•â•â•â•â•â•â•â•â•â•â•â•â•â•â•â•â•â•
       IF #EmergencyStop AND #BtnStop AND NOT #BtnStart AND NOT #Running THEN
           #Running := TRUE;   // Auto-start when safe
       END_IF;
       IF #BtnStart AND NOT #Running AND #EmergencyStop THEN
           #Running := TRUE;
       END_IF;

       IF NOT #BtnStop OR NOT #EmergencyStop THEN
           #Running := FALSE;
       END_IF;

       IF #BtnReset THEN
           #Running := FALSE;
           #iState := 0;
           #TargetFloor := 0;
           #DwellTimer := 0;
           #ItemCount := 0;
           #Up := FALSE;
           #Down := FALSE;
           #Slow := FALSE;
           #Load := FALSE;
           #Unload := FALSE;
           #ResetLight := TRUE;
           #StartLight := FALSE;
           #StopLight := FALSE;
           RETURN;
       END_IF;

       // â•â•â•â•â•â•â•â•â•â•â•â•â•â•â•â•â•â•â•â•â•â•â•â•â•â•â•â•â•â•â•â•â•â•â•â•â•â•â•â•â•â•â•â•â•â•â•â•â•â•â•â•
       // Panel indicator lights
       // â•â•â•â•â•â•â•â•â•â•â•â•â•â•â•â•â•â•â•â•â•â•â•â•â•â•â•â•â•â•â•â•â•â•â•â•â•â•â•â•â•â•â•â•â•â•â•â•â•â•â•â•
       #StartLight := #Running;
       #StopLight := NOT #Running;
       #ResetLight := FALSE;

       // â•â•â•â•â•â•â•â•â•â•â•â•â•â•â•â•â•â•â•â•â•â•â•â•â•â•â•â•â•â•â•â•â•â•â•â•â•â•â•â•â•â•â•â•â•â•â•â•â•â•â•â•
       // Track current floor from position sensors
       // High sensor = elevator platform aligned at floor level
       // Low sensor = approaching floor (triggered first)
       // Use High sensor as the primary floor-aligned indicator
       // â•â•â•â•â•â•â•â•â•â•â•â•â•â•â•â•â•â•â•â•â•â•â•â•â•â•â•â•â•â•â•â•â•â•â•â•â•â•â•â•â•â•â•â•â•â•â•â•â•â•â•â•
       IF #At0High THEN
           #CurrentFloor := 0;
       END_IF;
       IF #At1High THEN
           #CurrentFloor := 1;
       END_IF;
       IF #At2High THEN
           #CurrentFloor := 2;
       END_IF;
       IF #At3High THEN
           #CurrentFloor := 3;
       END_IF;

       // Floor indicator lights
       #Floor1Ind := (#CurrentFloor = 1);
       #Floor2Ind := (#CurrentFloor = 2);
       #Floor3Ind := (#CurrentFloor = 3);

       // Display shows items collected in current box
       #Display := INT_TO_DINT(#ItemCount);

       // â•â•â•â•â•â•â•â•â•â•â•â•â•â•â•â•â•â•â•â•â•â•â•â•â•â•â•â•â•â•â•â•â•â•â•â•â•â•â•â•â•â•â•â•â•â•â•â•â•â•â•â•
       // NOT running â†’ stop everything
       // â•â•â•â•â•â•â•â•â•â•â•â•â•â•â•â•â•â•â•â•â•â•â•â•â•â•â•â•â•â•â•â•â•â•â•â•â•â•â•â•â•â•â•â•â•â•â•â•â•â•â•â•
       IF NOT #Running THEN
           #Up := FALSE;
           #Down := FALSE;
           #Slow := FALSE;
           #Load := FALSE;
           #Unload := FALSE;
           #Conveyor0 := FALSE;
           #Conveyor1 := FALSE;
           #Conveyor2 := FALSE;
           #Conveyor3 := FALSE;
           #ExitConveyor := FALSE;
           #WarningLight := FALSE;
           #Green1 := FALSE;
           #Yellow1 := TRUE;
           #Red1 := FALSE;
           #Green2 := FALSE;
           #Yellow2 := TRUE;
           #Red2 := FALSE;
           #Green3 := FALSE;
           #Yellow3 := TRUE;
           #Red3 := FALSE;
           RETURN;
       END_IF;

       // â•â•â•â•â•â•â•â•â•â•â•â•â•â•â•â•â•â•â•â•â•â•â•â•â•â•â•â•â•â•â•â•â•â•â•â•â•â•â•â•â•â•â•â•â•â•â•â•â•â•â•â•
       // RUNNING â€” Floor conveyors 1-3 always ON (items advance to pickup)
       // Conveyor0 and ExitConveyor controlled by state machine
       // â•â•â•â•â•â•â•â•â•â•â•â•â•â•â•â•â•â•â•â•â•â•â•â•â•â•â•â•â•â•â•â•â•â•â•â•â•â•â•â•â•â•â•â•â•â•â•â•â•â•â•â•
       #Conveyor1 := TRUE;
       #Conveyor2 := TRUE;
       #Conveyor3 := TRUE;

       // â•â•â•â•â•â•â•â•â•â•â•â•â•â•â•â•â•â•â•â•â•â•â•â•â•â•â•â•â•â•â•â•â•â•â•â•â•â•â•â•â•â•â•â•â•â•â•â•â•â•â•â•
       // Elevator state machine â€” collect MaxItems items into box
       //   S0 = LOAD_BOX:  At floor 0, wait for box from emitter, load onto elevator
       //   S1 = SCAN:      Check floors 1-3 for waiting items
       //   S2 = MOVING:    Go to target floor
       //   S3 = COLLECT:   At target floor, load item into box on elevator
       //   S4 = RETURN:    Box full, go back to floor 0
       //   S5 = UNLOAD:    At floor 0, push full box off elevator
       //
       // Floor arrival: use High sensor only (robust against overshoot)
       // Floor approach: use Low sensor (triggers before High)
       // â•â•â•â•â•â•â•â•â•â•â•â•â•â•â•â•â•â•â•â•â•â•â•â•â•â•â•â•â•â•â•â•â•â•â•â•â•â•â•â•â•â•â•â•â•â•â•â•â•â•â•â•
       CASE #iState OF
           0: // LOAD_BOX â€” at floor 0, wait for empty box, load it
               #Unload := FALSE;
               #WarningLight := FALSE;
               #ExitConveyor := FALSE;

               // First ensure we're at floor 0
               IF NOT #At0High THEN
                   // Not at floor 0 â€” drive down
                   #Load := FALSE;
                   #Conveyor0 := FALSE;
                   IF #At0Low THEN
                       #Down := TRUE;
                       #Up := FALSE;
                       #Slow := TRUE;
                   ELSE
                       #Down := TRUE;
                       #Up := FALSE;
                       #Slow := FALSE;
                   END_IF;
               ELSE
                   // At floor 0 â€” run conveyor to bring box, activate Load
                   #Up := FALSE;
                   #Down := FALSE;
                   #Slow := FALSE;
                   #Conveyor0 := TRUE;
                   #Load := TRUE;
                   #DwellTimer := #DwellTimer + 1;

                   // AtElevator = box/item on elevator platform
                   // Wait at least 200 scans (~2s) for box to settle on platform
                   IF #AtElevator AND #DwellTimer > 200 THEN
                       // Box is on elevator and settled
                       #Load := FALSE;
                       #Conveyor0 := FALSE;
                       #ItemCount := 0;
                       #DwellTimer := 0;
                       #iState := 1;
                   END_IF;

                   // Safety timeout: if no box after long wait, keep trying
                   IF #DwellTimer > 1000 THEN
                       #DwellTimer := 0;
                   END_IF;
               END_IF;

           1: // SCAN â€” check which floors have items waiting
               #Up := FALSE;
               #Down := FALSE;
               #Slow := FALSE;
               #Load := FALSE;
               #Unload := FALSE;
               #WarningLight := FALSE;
               #Conveyor0 := FALSE;
               #ExitConveyor := FALSE;

               // Priority scan: floor 1 â†’ 2 â†’ 3
               IF #At1 THEN
                   #TargetFloor := 1;
                   #DwellTimer := 0;
                   #iState := 2;
               ELSIF #At2 THEN
                   #TargetFloor := 2;
                   #DwellTimer := 0;
                   #iState := 2;
               ELSIF #At3 THEN
                   #TargetFloor := 3;
                   #DwellTimer := 0;
                   #iState := 2;
               END_IF;
               // If no items waiting, keep scanning â€” emitters will spawn items

           2: // MOVING â€” go to target floor
               #Load := FALSE;
               #Unload := FALSE;
               #Conveyor0 := FALSE;
               #ExitConveyor := FALSE;
               #WarningLight := TRUE;

               // Check position using High sensor for arrival, Low for approach
               CASE #TargetFloor OF
                   0:
                       #atTarget := #At0High;
                       #nearTarget := #At0Low AND NOT #At0High;
                   1:
                       #atTarget := #At1High;
                       #nearTarget := #At1Low AND NOT #At1High;
                   2:
                       #atTarget := #At2High;
                       #nearTarget := #At2Low AND NOT #At2High;
                   3:
                       #atTarget := #At3High;
                       #nearTarget := #At3Low AND NOT #At3High;
               END_CASE;

               IF #atTarget THEN
                   // Arrived at target floor â€” stop immediately
                   #Up := FALSE;
                   #Down := FALSE;
                   #Slow := FALSE;
                   #WarningLight := FALSE;
                   #DwellTimer := 0;
                   #iState := 3;
               ELSIF #nearTarget THEN
                   // Approaching â€” slow down, keep same direction
                   #Slow := TRUE;
                   IF #CurrentFloor < #TargetFloor THEN
                       #Up := TRUE;
                       #Down := FALSE;
                   ELSE
                       #Up := FALSE;
                       #Down := TRUE;
                   END_IF;
               ELSE
                   // Far from target â€” full speed
                   #Slow := FALSE;
                   IF #CurrentFloor < #TargetFloor THEN
                       #Up := TRUE;
                       #Down := FALSE;
                   ELSE
                       #Up := FALSE;
                       #Down := TRUE;
                   END_IF;
               END_IF;

           3: // COLLECT â€” at target floor, load item into box
               #Up := FALSE;
               #Down := FALSE;
               #Slow := FALSE;
               #Unload := FALSE;
               #WarningLight := FALSE;

               // Run the floor conveyor to push item toward elevator + Load
               CASE #TargetFloor OF
                   1:
                       #Conveyor1 := TRUE;
                   2:
                       #Conveyor2 := TRUE;
                   3:
                       #Conveyor3 := TRUE;
               END_CASE;
               #Load := TRUE;

               #DwellTimer := #DwellTimer + 1;

               // Fixed dwell: 400 scans (~4 seconds) for reliable physical transfer
               // This ensures the item physically moves from floor conveyor into box
               IF #DwellTimer > 400 THEN
                   #Load := FALSE;
                   #ItemCount := #ItemCount + 1;
                   #DwellTimer := 0;

                   // Check if box is full
                   IF #ItemCount >= #MaxItems THEN
                       // Box full â€” go unload at floor 0
                       #TargetFloor := 0;
                       #iState := 4;
                   ELSE
                       // Need more items â€” rescan
                       #iState := 1;
                   END_IF;
               END_IF;

           4: // RETURN â€” full box, go back to floor 0
               #Load := FALSE;
               #Unload := FALSE;
               #Conveyor0 := FALSE;
               #ExitConveyor := FALSE;
               #WarningLight := TRUE;

               #atTarget := #At0High;
               #nearTarget := #At0Low AND NOT #At0High;

               IF #atTarget THEN
                   // Arrived at floor 0
                   #Up := FALSE;
                   #Down := FALSE;
                   #Slow := FALSE;
                   #WarningLight := FALSE;
                   #DwellTimer := 0;
                   #iState := 5;
               ELSIF #nearTarget THEN
                   #Up := FALSE;
                   #Down := TRUE;
                   #Slow := TRUE;
               ELSE
                   #Up := FALSE;
                   #Down := TRUE;
                   #Slow := FALSE;
               END_IF;

           5: // UNLOAD â€” push full box off at floor 0
               #Up := FALSE;
               #Down := FALSE;
               #Slow := FALSE;
               #Load := FALSE;
               #Unload := TRUE;
               #Conveyor0 := TRUE;
               #ExitConveyor := TRUE;
               #WarningLight := FALSE;

               #DwellTimer := #DwellTimer + 1;

               // Wait for box to leave elevator platform
               // Min 300 scans (~3s) to ensure box physically exits
               IF (NOT #AtElevator AND #DwellTimer > 300) OR (#DwellTimer > 500) THEN
                   #Unload := FALSE;
                   #Conveyor0 := FALSE;
                   #ExitConveyor := FALSE;
                   #DwellTimer := 0;
                   #ItemCount := 0;
                   #iState := 0;  // Go load next empty box
               END_IF;

           ELSE
               #iState := 0;
       END_CASE;

       // â•â•â•â•â•â•â•â•â•â•â•â•â•â•â•â•â•â•â•â•â•â•â•â•â•â•â•â•â•â•â•â•â•â•â•â•â•â•â•â•â•â•â•â•â•â•â•â•â•â•â•â•
       // Traffic lights per floor (1-3)
       //   Green  = elevator at this floor, collecting item
       //   Yellow = elevator approaching this floor
       //   Red    = elevator busy elsewhere
       // â•â•â•â•â•â•â•â•â•â•â•â•â•â•â•â•â•â•â•â•â•â•â•â•â•â•â•â•â•â•â•â•â•â•â•â•â•â•â•â•â•â•â•â•â•â•â•â•â•â•â•â•
       // Floor 1
       #Green1 := (#CurrentFloor = 1) AND (#iState = 3);
       #Yellow1 := (#TargetFloor = 1) AND (#iState = 2) AND (#At1Low OR #At1High);
       #Red1 := NOT #Green1 AND NOT #Yellow1 AND ((#iState = 2) OR (#iState = 4));

       // Floor 2
       #Green2 := (#CurrentFloor = 2) AND (#iState = 3);
       #Yellow2 := (#TargetFloor = 2) AND (#iState = 2) AND (#At2Low OR #At2High);
       #Red2 := NOT #Green2 AND NOT #Yellow2 AND ((#iState = 2) OR (#iState = 4));

       // Floor 3
       #Green3 := (#CurrentFloor = 3) AND (#iState = 3);
       #Yellow3 := (#TargetFloor = 3) AND (#iState = 2) AND (#At3Low OR #At3High);
       #Red3 := NOT #Green3 AND NOT #Yellow3 AND ((#iState = 2) OR (#iState = 4));
END_FUNCTION_BLOCK

FUNCTION_BLOCK "FB_ElevatorBasic"   // FB7, SCL
{ S7_Optimized_Access := 'FALSE' }
VERSION : 0.4
// MANTIS â€” Scene 11: Elevator (Basic)
//  Two elevators transport items through 3 levels (0, 1, 2).
//  Left elevator shuttles Level 0 â†” Level 1.
//  Right elevator shuttles Level 1 â†” Level 2.
//  DB20: Instance DB (non-optimized access)
// 
//  Factory I/O layout:
//    3-level structure with left and right elevator shafts.
//    Entry conveyor feeds items at level 0.
//    Left elevator carries items from level 0 â†’ level 1.
//    Right elevator carries items from level 1 â†’ level 2.
//    Exit conveyor removes items at level 2.
//    Load/Unload conveyors at each elevator stop.
//    Traffic lights (3 sets) and warning lights for safety.
//    Start/Stop/Reset/EmergencyStop/Auto buttons on control panel.
// 
//  Driver mapping (from Factory I/O):
//    SENSORS (Inputs):
//      NOTE: Use %I10.x-%I13.x (NOT %I0.x-%I3.x) because the PLC's
//      built-in physical DI module owns %IB0/%IB1 and overwrites external writes.
//      At entry        â†’ %I10.0   At entry left    â†’ %I10.1
//      At exit left    â†’ %I10.2   At entry 0       â†’ %I10.3
//      At exit 0       â†’ %I10.4   At entry right   â†’ %I10.5
//      At exit right   â†’ %I10.6   At exit          â†’ %I10.7
//      At entry 1      â†’ %I11.0   At exit 1        â†’ %I11.1
//      At entry 2      â†’ %I11.2   At exit 2        â†’ %I11.3
//      At left low 0   â†’ %I11.4   At left high 0   â†’ %I11.5
//      At left low 1   â†’ %I11.6   At left high 1   â†’ %I11.7
//      At left low 2   â†’ %I12.0   At left high 2   â†’ %I12.1
//      At right low 0  â†’ %I12.2   At right high 0  â†’ %I12.3
//      At right low 1  â†’ %I12.4   At right high 1  â†’ %I12.5
//      At right low 2  â†’ %I12.6   At right high 2  â†’ %I12.7
//      Start           â†’ %I13.0   Reset            â†’ %I13.1
//      Stop            â†’ %I13.2   Emergency stop   â†’ %I13.3
//      Auto            â†’ %I13.4   FACTORY I/O (Running) â†’ %I13.5
// 
//    ACTUATORS (Outputs):
//      Entry conveyor  â†’ %Q0.0    Unload left      â†’ %Q0.1
//      Load left       â†’ %Q0.2    Conveyor 0       â†’ %Q0.3
//      Unload right    â†’ %Q0.4    Load right       â†’ %Q0.5
//      Exit conveyor   â†’ %Q0.6    Left up          â†’ %Q0.7
//      Left slow       â†’ %Q1.0    Left down        â†’ %Q1.1
//      Right up        â†’ %Q1.2    Right slow       â†’ %Q1.3
//      Right down      â†’ %Q1.4    Conveyor 1       â†’ %Q1.5
//      Conveyor 2      â†’ %Q1.6    Left warning     â†’ %Q1.7
//      Right warning   â†’ %Q2.0    Green 0          â†’ %Q2.1
//      Yellow 0        â†’ %Q2.2    Red 0            â†’ %Q2.3
//      B green         â†’ %Q2.4    B yellow         â†’ %Q2.5
//      B red           â†’ %Q2.6    C green          â†’ %Q2.7
//      C yellow        â†’ %Q3.0    C red            â†’ %Q3.1
//      Start light     â†’ %Q3.2    Reset light      â†’ %Q3.3
//      Stop light      â†’ %Q3.4
// 
//  DB20 byte layout (non-optimized, BOOL = 2 bytes):
//    Sensors:
//      0:  AtEntry          2:  AtEntryLeft      4:  AtExitLeft
//      6:  AtEntry0         8:  AtExit0         10:  AtEntryRight
//     12:  AtExitRight     14:  AtExit          16:  AtEntry1
//     18:  AtExit1         20:  AtEntry2        22:  AtExit2
//     24:  AtLeftLow0      26:  AtLeftHigh0     28:  AtLeftLow1
//     30:  AtLeftHigh1     32:  AtLeftLow2      34:  AtLeftHigh2
//     36:  AtRightLow0     38:  AtRightHigh0    40:  AtRightLow1
//     42:  AtRightHigh1    44:  AtRightLow2     46:  AtRightHigh2
//     48:  BtnStart        50:  BtnReset        52:  BtnStop
//     54:  EmergencyStop   56:  BtnAuto
//    Actuators:
//     58:  EntryConveyor   60:  UnloadLeft      62:  LoadLeft
//     64:  Conveyor0       66:  UnloadRight     68:  LoadRight
//     70:  ExitConveyor    72:  LeftUp          74:  LeftSlow
//     76:  LeftDown        78:  RightUp         80:  RightSlow
//     82:  RightDown       84:  Conveyor1       86:  Conveyor2
//     88:  LeftWarning     90:  RightWarning    92:  Green0
//     94:  Yellow0         96:  Red0            98:  BGreen
//    100:  BYellow        102:  BRed           104:  CGreen
//    106:  CYellow        108:  CRed           110:  StartLight
//    112:  ResetLight     114:  StopLight
//    Internal:
//    116:  LeftState (INT)  118: RightState (INT)
//    120:  LeftTimer (INT)  122: RightTimer (INT)
//    124:  Running (BOOL)   126: Enable (BOOL)
//    Total = 128 bytes
// 
//  Vulnerability: Enable (byte 126, default TRUE) is read by logic
//    but NEVER written. Setting Enable=FALSE stops all elevators
//    and conveyors permanently.
//  â”€â”€ Sensors (inputs) â”€â”€
   VAR
      AtEntry : Bool;   // byte 0 â€” %I10.0
      _p00 : Byte;
      AtEntryLeft : Bool;   // byte 2 â€” %I10.1
      _p01 : Byte;
      AtExitLeft : Bool;   // byte 4 â€” %I10.2
      _p02 : Byte;
      AtEntry0 : Bool;   // byte 6 â€” %I10.3
      _p03 : Byte;
      AtExit0 : Bool;   // byte 8 â€” %I10.4
      _p04 : Byte;
      AtEntryRight : Bool;   // byte 10 â€” %I10.5
      _p05 : Byte;
      AtExitRight : Bool;   // byte 12 â€” %I10.6
      _p06 : Byte;
      AtExit : Bool;   // byte 14 â€” %I10.7
      _p07 : Byte;
      AtEntry1 : Bool;   // byte 16 â€” %I11.0
      _p08 : Byte;
      AtExit1 : Bool;   // byte 18 â€” %I11.1
      _p09 : Byte;
      AtEntry2 : Bool;   // byte 20 â€” %I11.2
      _p10 : Byte;
      AtExit2 : Bool;   // byte 22 â€” %I11.3
      _p11 : Byte;
      AtLeftLow0 : Bool;   // byte 24 â€” %I11.4
      _p12 : Byte;
      AtLeftHigh0 : Bool;   // byte 26 â€” %I11.5
      _p13 : Byte;
      AtLeftLow1 : Bool;   // byte 28 â€” %I11.6
      _p14 : Byte;
      AtLeftHigh1 : Bool;   // byte 30 â€” %I11.7
      _p15 : Byte;
      AtLeftLow2 : Bool;   // byte 32 â€” %I12.0
      _p16 : Byte;
      AtLeftHigh2 : Bool;   // byte 34 â€” %I12.1
      _p17 : Byte;
      AtRightLow0 : Bool;   // byte 36 â€” %I12.2
      _p18 : Byte;
      AtRightHigh0 : Bool;   // byte 38 â€” %I12.3
      _p19 : Byte;
      AtRightLow1 : Bool;   // byte 40 â€” %I12.4
      _p20 : Byte;
      AtRightHigh1 : Bool;   // byte 42 â€” %I12.5
      _p21 : Byte;
      AtRightLow2 : Bool;   // byte 44 â€” %I12.6
      _p22 : Byte;
      AtRightHigh2 : Bool;   // byte 46 â€” %I12.7
      _p23 : Byte;
      BtnStart : Bool;   // byte 48 â€” %I13.0
      _p24 : Byte;
      BtnReset : Bool;   // byte 50 â€” %I13.1
      _p25 : Byte;
      BtnStop : Bool;   // byte 52 â€” %I13.2
      _p26 : Byte;
      EmergencyStop : Bool;   // byte 54 â€” %I13.3
      _p27 : Byte;
      BtnAuto : Bool;   // byte 56 â€” %I13.4
      _p28 : Byte;   // â”€â”€ Actuators (outputs) â”€â”€
      EntryConveyor : Bool;   // byte 58 â€” %Q0.0
      _p29 : Byte;
      UnloadLeft : Bool;   // byte 60 â€” %Q0.1
      _p30 : Byte;
      LoadLeft : Bool;   // byte 62 â€” %Q0.2
      _p31 : Byte;
      Conveyor0 : Bool;   // byte 64 â€” %Q0.3
      _p32 : Byte;
      UnloadRight : Bool;   // byte 66 â€” %Q0.4
      _p33 : Byte;
      LoadRight : Bool;   // byte 68 â€” %Q0.5
      _p34 : Byte;
      ExitConveyor : Bool;   // byte 70 â€” %Q0.6
      _p35 : Byte;
      LeftUp : Bool;   // byte 72 â€” %Q0.7
      _p36 : Byte;
      LeftSlow : Bool;   // byte 74 â€” %Q1.0
      _p37 : Byte;
      LeftDown : Bool;   // byte 76 â€” %Q1.1
      _p38 : Byte;
      RightUp : Bool;   // byte 78 â€” %Q1.2
      _p39 : Byte;
      RightSlow : Bool;   // byte 80 â€” %Q1.3
      _p40 : Byte;
      RightDown : Bool;   // byte 82 â€” %Q1.4
      _p41 : Byte;
      Conveyor1 : Bool;   // byte 84 â€” %Q1.5
      _p42 : Byte;
      Conveyor2 : Bool;   // byte 86 â€” %Q1.6
      _p43 : Byte;
      LeftWarning : Bool;   // byte 88 â€” %Q1.7
      _p44 : Byte;
      RightWarning : Bool;   // byte 90 â€” %Q2.0
      _p45 : Byte;
      Green0 : Bool;   // byte 92 â€” %Q2.1
      _p46 : Byte;
      Yellow0 : Bool;   // byte 94 â€” %Q2.2
      _p47 : Byte;
      Red0 : Bool;   // byte 96 â€” %Q2.3
      _p48 : Byte;
      BGreen : Bool;   // byte 98 â€” %Q2.4
      _p49 : Byte;
      BYellow : Bool;   // byte 100 â€” %Q2.5
      _p50 : Byte;
      BRed : Bool;   // byte 102 â€” %Q2.6
      _p51 : Byte;
      CGreen : Bool;   // byte 104 â€” %Q2.7
      _p52 : Byte;
      CYellow : Bool;   // byte 106 â€” %Q3.0
      _p53 : Byte;
      CRed : Bool;   // byte 108 â€” %Q3.1
      _p54 : Byte;
      StartLight : Bool;   // byte 110 â€” %Q3.2
      _p55 : Byte;
      ResetLight : Bool;   // byte 112 â€” %Q3.3
      _p56 : Byte;
      StopLight : Bool;   // byte 114 â€” %Q3.4
      _p57 : Byte;   // â”€â”€ Internal state â”€â”€
      LeftState : Int := 0;   // byte 116 â€” left elevator state machine
      RightState : Int := 0;   // byte 118 â€” right elevator state machine
      LeftTimer : Int := 0;   // byte 120 â€” left elevator dwell timer
      RightTimer : Int := 0;   // byte 122 â€” right elevator dwell timer
      Running : Bool := FALSE;   // byte 124 â€” system running
      _p58 : Byte;
      Enable : Bool := TRUE;   // byte 126 â€” system enable (default ON)
      _p59 : Byte;   // Total: 128 bytes
   END_VAR
BEGIN
       // â•â•â•â•â•â•â•â•â•â•â•â•â•â•â•â•â•â•â•â•â•â•â•â•â•â•â•â•â•â•â•â•â•â•â•â•â•â•â•â•â•â•â•â•â•â•â•â•â•â•â•â•
       // Safety gate: if Enable is FALSE, shut everything down
       // â•â•â•â•â•â•â•â•â•â•â•â•â•â•â•â•â•â•â•â•â•â•â•â•â•â•â•â•â•â•â•â•â•â•â•â•â•â•â•â•â•â•â•â•â•â•â•â•â•â•â•â•
       IF NOT #Enable THEN
           #Running := FALSE;
           // Stop elevators
           #LeftUp := FALSE;
           #LeftSlow := FALSE;
           #LeftDown := FALSE;
           #RightUp := FALSE;
           #RightSlow := FALSE;
           #RightDown := FALSE;
           // Stop conveyors
           #EntryConveyor := FALSE;
           #ExitConveyor := FALSE;
           #Conveyor0 := FALSE;
           #Conveyor1 := FALSE;
           #Conveyor2 := FALSE;
           #LoadLeft := FALSE;
           #UnloadLeft := FALSE;
           #LoadRight := FALSE;
           #UnloadRight := FALSE;
           // Warnings ON, all traffic lights RED
           #LeftWarning := TRUE;
           #RightWarning := TRUE;
           #Green0 := FALSE;
           #Yellow0 := FALSE;
           #Red0 := TRUE;
           #BGreen := FALSE;
           #BYellow := FALSE;
           #BRed := TRUE;
           #CGreen := FALSE;
           #CYellow := FALSE;
           #CRed := TRUE;
           // Panel lights
           #StartLight := FALSE;
           #ResetLight := FALSE;
           #StopLight := TRUE;
           RETURN;
       END_IF;

       // â•â•â•â•â•â•â•â•â•â•â•â•â•â•â•â•â•â•â•â•â•â•â•â•â•â•â•â•â•â•â•â•â•â•â•â•â•â•â•â•â•â•â•â•â•â•â•â•â•â•â•â•
       // Button handling
       //
       // Factory I/O button conventions:
       //   Start  â†’ momentary, normally OPEN   (FALSE=idle, TRUE=pressed)
       //   Stop   â†’ momentary, normally CLOSED (TRUE=idle, FALSE=pressed)
       //   Reset  â†’ momentary, normally OPEN   (FALSE=idle, TRUE=pressed)
       //   E-Stop â†’ latching,  normally CLOSED (TRUE=normal, FALSE=engaged)
       //   Auto   â†’ selector switch
       // â•â•â•â•â•â•â•â•â•â•â•â•â•â•â•â•â•â•â•â•â•â•â•â•â•â•â•â•â•â•â•â•â•â•â•â•â•â•â•â•â•â•â•â•â•â•â•â•â•â•â•â•
       IF #BtnStart AND NOT #Running AND #EmergencyStop THEN
           #Running := TRUE;
       END_IF;

       IF NOT #BtnStop OR NOT #EmergencyStop THEN
           #Running := FALSE;
       END_IF;

       // Auto-start: if E-stop normal AND Stop not pressed, start automatically
       IF #EmergencyStop AND #BtnStop AND NOT #BtnStart THEN
           #Running := TRUE;
       END_IF;

       IF #BtnReset THEN
           #Running := FALSE;
           #LeftState := 0;
           #RightState := 0;
           #LeftTimer := 0;
           #RightTimer := 0;
           // Stop elevators
           #LeftUp := FALSE;
           #LeftSlow := FALSE;
           #LeftDown := FALSE;
           #RightUp := FALSE;
           #RightSlow := FALSE;
           #RightDown := FALSE;
           // Stop conveyors
           #EntryConveyor := FALSE;
           #ExitConveyor := FALSE;
           #Conveyor0 := FALSE;
           #Conveyor1 := FALSE;
           #Conveyor2 := FALSE;
           #LoadLeft := FALSE;
           #UnloadLeft := FALSE;
           #LoadRight := FALSE;
           #UnloadRight := FALSE;
           // Lights
           #ResetLight := TRUE;
           #StartLight := FALSE;
           #StopLight := FALSE;
           #LeftWarning := FALSE;
           #RightWarning := FALSE;
           #Green0 := FALSE;
           #Yellow0 := TRUE;
           #Red0 := FALSE;
           #BGreen := FALSE;
           #BYellow := TRUE;
           #BRed := FALSE;
           #CGreen := FALSE;
           #CYellow := TRUE;
           #CRed := FALSE;
           RETURN;
       END_IF;

       // â•â•â•â•â•â•â•â•â•â•â•â•â•â•â•â•â•â•â•â•â•â•â•â•â•â•â•â•â•â•â•â•â•â•â•â•â•â•â•â•â•â•â•â•â•â•â•â•â•â•â•â•
       // Panel indicator lights
       // â•â•â•â•â•â•â•â•â•â•â•â•â•â•â•â•â•â•â•â•â•â•â•â•â•â•â•â•â•â•â•â•â•â•â•â•â•â•â•â•â•â•â•â•â•â•â•â•â•â•â•â•
       #StartLight := #Running;
       #StopLight := NOT #Running;
       #ResetLight := FALSE;

       // â•â•â•â•â•â•â•â•â•â•â•â•â•â•â•â•â•â•â•â•â•â•â•â•â•â•â•â•â•â•â•â•â•â•â•â•â•â•â•â•â•â•â•â•â•â•â•â•â•â•â•â•
       // NOT running â†’ all outputs OFF
       // â•â•â•â•â•â•â•â•â•â•â•â•â•â•â•â•â•â•â•â•â•â•â•â•â•â•â•â•â•â•â•â•â•â•â•â•â•â•â•â•â•â•â•â•â•â•â•â•â•â•â•â•
       IF NOT #Running THEN
           #LeftUp := FALSE;
           #LeftSlow := FALSE;
           #LeftDown := FALSE;
           #RightUp := FALSE;
           #RightSlow := FALSE;
           #RightDown := FALSE;
           #EntryConveyor := FALSE;
           #ExitConveyor := FALSE;
           #Conveyor0 := FALSE;
           #Conveyor1 := FALSE;
           #Conveyor2 := FALSE;
           #LoadLeft := FALSE;
           #UnloadLeft := FALSE;
           #LoadRight := FALSE;
           #UnloadRight := FALSE;
           #LeftWarning := FALSE;
           #RightWarning := FALSE;
           #Green0 := FALSE;
           #Yellow0 := TRUE;
           #Red0 := FALSE;
           #BGreen := FALSE;
           #BYellow := TRUE;
           #BRed := FALSE;
           #CGreen := FALSE;
           #CYellow := TRUE;
           #CRed := FALSE;
           RETURN;
       END_IF;

       // â•â•â•â•â•â•â•â•â•â•â•â•â•â•â•â•â•â•â•â•â•â•â•â•â•â•â•â•â•â•â•â•â•â•â•â•â•â•â•â•â•â•â•â•â•â•â•â•â•â•â•â•
       // RUNNING â€” Conveyors always ON
       // â•â•â•â•â•â•â•â•â•â•â•â•â•â•â•â•â•â•â•â•â•â•â•â•â•â•â•â•â•â•â•â•â•â•â•â•â•â•â•â•â•â•â•â•â•â•â•â•â•â•â•â•
       #EntryConveyor := TRUE;
       #ExitConveyor := TRUE;
       #Conveyor0 := TRUE;
       #Conveyor1 := TRUE;
       #Conveyor2 := TRUE;

       // â•â•â•â•â•â•â•â•â•â•â•â•â•â•â•â•â•â•â•â•â•â•â•â•â•â•â•â•â•â•â•â•â•â•â•â•â•â•â•â•â•â•â•â•â•â•â•â•â•â•â•â•
       // LEFT ELEVATOR â€” Level 0 â†” Level 1
       // State 0: At Level 0, loading (wait for item)
       // State 1: Going up to Level 1
       // State 2: At Level 1, unloading (dwell timer)
       // State 3: Going down to Level 0
       // â•â•â•â•â•â•â•â•â•â•â•â•â•â•â•â•â•â•â•â•â•â•â•â•â•â•â•â•â•â•â•â•â•â•â•â•â•â•â•â•â•â•â•â•â•â•â•â•â•â•â•â•
       CASE #LeftState OF
           0: // At Level 0 â€” load item onto elevator
               #LeftUp := FALSE;
               #LeftSlow := FALSE;
               #LeftDown := FALSE;
               #LoadLeft := TRUE;       // Elevator rollers pull item in
               #UnloadLeft := FALSE;
               #LeftWarning := FALSE;
               IF #AtEntryLeft THEN
                   #LeftTimer := #LeftTimer + 1;
                   IF #LeftTimer > 50 THEN   // ~500ms dwell for loading
                       #LeftTimer := 0;
                       #LoadLeft := FALSE;
                       #LeftState := 1;
                   END_IF;
               ELSE
                   #LeftTimer := 0;
               END_IF;

           1: // Going up to Level 1
               #LoadLeft := FALSE;
               #UnloadLeft := FALSE;
               #LeftWarning := TRUE;
               // Dual-sensor: BOTH = at floor, EITHER = approaching
               IF #AtLeftLow1 AND #AtLeftHigh1 THEN
                   // Arrived at Level 1
                   #LeftUp := FALSE;
                   #LeftDown := FALSE;
                   #LeftSlow := FALSE;
                   #LeftTimer := 0;
                   #LeftState := 2;
               ELSIF #AtLeftLow1 OR #AtLeftHigh1 THEN
                   // Approaching â€” slow down
                   #LeftUp := TRUE;
                   #LeftDown := FALSE;
                   #LeftSlow := TRUE;
               ELSE
                   // Far â€” full speed
                   #LeftUp := TRUE;
                   #LeftDown := FALSE;
                   #LeftSlow := FALSE;
               END_IF;

           2: // At Level 1 â€” unload item off elevator
               #LeftUp := FALSE;
               #LeftSlow := FALSE;
               #LeftDown := FALSE;
               #LoadLeft := FALSE;
               #UnloadLeft := TRUE;     // Elevator rollers push item out
               #LeftWarning := FALSE;
               #LeftTimer := #LeftTimer + 1;
               IF #LeftTimer > 100 THEN      // ~1s dwell for unloading
                   #LeftTimer := 0;
                   #UnloadLeft := FALSE;
                   #LeftState := 3;
               END_IF;

           3: // Going down to Level 0
               #UnloadLeft := FALSE;
               #LoadLeft := FALSE;
               #LeftWarning := TRUE;
               // Dual-sensor position detection
               IF #AtLeftLow0 AND #AtLeftHigh0 THEN
                   // Arrived at Level 0
                   #LeftUp := FALSE;
                   #LeftDown := FALSE;
                   #LeftSlow := FALSE;
                   #LeftState := 0;
               ELSIF #AtLeftLow0 OR #AtLeftHigh0 THEN
                   // Approaching â€” slow down
                   #LeftUp := FALSE;
                   #LeftDown := TRUE;
                   #LeftSlow := TRUE;
               ELSE
                   // Far â€” full speed
                   #LeftUp := FALSE;
                   #LeftDown := TRUE;
                   #LeftSlow := FALSE;
               END_IF;

           ELSE
               #LeftState := 0;
       END_CASE;

       // â•â•â•â•â•â•â•â•â•â•â•â•â•â•â•â•â•â•â•â•â•â•â•â•â•â•â•â•â•â•â•â•â•â•â•â•â•â•â•â•â•â•â•â•â•â•â•â•â•â•â•â•
       // RIGHT ELEVATOR â€” Level 1 â†” Level 2
       // State 0: At Level 1, loading (wait for item)
       // State 1: Going up to Level 2
       // State 2: At Level 2, unloading (dwell timer)
       // State 3: Going down to Level 1
       // â•â•â•â•â•â•â•â•â•â•â•â•â•â•â•â•â•â•â•â•â•â•â•â•â•â•â•â•â•â•â•â•â•â•â•â•â•â•â•â•â•â•â•â•â•â•â•â•â•â•â•â•
       CASE #RightState OF
           0: // At Level 1 â€” load item onto elevator
               #RightUp := FALSE;
               #RightSlow := FALSE;
               #RightDown := FALSE;
               #LoadRight := TRUE;      // Elevator rollers pull item in
               #UnloadRight := FALSE;
               #RightWarning := FALSE;
               IF #AtEntryRight THEN
                   #RightTimer := #RightTimer + 1;
                   IF #RightTimer > 50 THEN   // ~500ms dwell for loading
                       #RightTimer := 0;
                       #LoadRight := FALSE;
                       #RightState := 1;
                   END_IF;
               ELSE
                   #RightTimer := 0;
               END_IF;

           1: // Going up to Level 2
               #LoadRight := FALSE;
               #UnloadRight := FALSE;
               #RightWarning := TRUE;
               // Dual-sensor: BOTH = at floor, EITHER = approaching
               IF #AtRightLow2 AND #AtRightHigh2 THEN
                   // Arrived at Level 2
                   #RightUp := FALSE;
                   #RightDown := FALSE;
                   #RightSlow := FALSE;
                   #RightTimer := 0;
                   #RightState := 2;
               ELSIF #AtRightLow2 OR #AtRightHigh2 THEN
                   // Approaching â€” slow down
                   #RightUp := TRUE;
                   #RightDown := FALSE;
                   #RightSlow := TRUE;
               ELSE
                   // Far â€” full speed
                   #RightUp := TRUE;
                   #RightDown := FALSE;
                   #RightSlow := FALSE;
               END_IF;

           2: // At Level 2 â€” unload item off elevator
               #RightUp := FALSE;
               #RightSlow := FALSE;
               #RightDown := FALSE;
               #LoadRight := FALSE;
               #UnloadRight := TRUE;    // Elevator rollers push item out
               #RightWarning := FALSE;
               #RightTimer := #RightTimer + 1;
               IF #RightTimer > 100 THEN     // ~1s dwell for unloading
                   #RightTimer := 0;
                   #UnloadRight := FALSE;
                   #RightState := 3;
               END_IF;

           3: // Going down to Level 1
               #UnloadRight := FALSE;
               #LoadRight := FALSE;
               #RightWarning := TRUE;
               // Dual-sensor position detection
               IF #AtRightLow1 AND #AtRightHigh1 THEN
                   // Arrived at Level 1
                   #RightUp := FALSE;
                   #RightDown := FALSE;
                   #RightSlow := FALSE;
                   #RightState := 0;
               ELSIF #AtRightLow1 OR #AtRightHigh1 THEN
                   // Approaching â€” slow down
                   #RightUp := FALSE;
                   #RightDown := TRUE;
                   #RightSlow := TRUE;
               ELSE
                   // Far â€” full speed
                   #RightUp := FALSE;
                   #RightDown := TRUE;
                   #RightSlow := FALSE;
               END_IF;

           ELSE
               #RightState := 0;
       END_CASE;

       // â•â•â•â•â•â•â•â•â•â•â•â•â•â•â•â•â•â•â•â•â•â•â•â•â•â•â•â•â•â•â•â•â•â•â•â•â•â•â•â•â•â•â•â•â•â•â•â•â•â•â•â•
       // Traffic lights
       //   Level 0: Green=safe, Yellow=approaching, Red=moving
       //   Level 1 (B): same
       //   Level 2 (C): same
       // â•â•â•â•â•â•â•â•â•â•â•â•â•â•â•â•â•â•â•â•â•â•â•â•â•â•â•â•â•â•â•â•â•â•â•â•â•â•â•â•â•â•â•â•â•â•â•â•â•â•â•â•
       // Level 0 lights â€” based on left elevator
       #Green0 := (#LeftState = 0);                         // Idle at level 0
       #Yellow0 := (#LeftState = 3) AND (#AtLeftLow0 OR #AtLeftHigh0);   // Approaching
       #Red0 := (#LeftState = 1) OR (#LeftState = 3);      // Moving

       // Level 1 lights (B) â€” both elevators interact here
       #BGreen := (#LeftState = 2) OR (#RightState = 0);     // Elevator at level 1
       #BYellow := ((#LeftState = 1) AND (#AtLeftLow1 OR #AtLeftHigh1))
       OR ((#RightState = 3) AND (#AtRightLow1 OR #AtRightHigh1));   // Approaching
       #BRed := (#LeftState = 1) OR (#LeftState = 3)
       OR (#RightState = 1) OR (#RightState = 3);    // Any moving

       // Level 2 lights (C) â€” based on right elevator
       #CGreen := (#RightState = 2);                        // At level 2
       #CYellow := (#RightState = 1) AND (#AtRightLow2 OR #AtRightHigh2);   // Approaching
       #CRed := (#RightState = 1) OR (#RightState = 3);   // Moving
END_FUNCTION_BLOCK

FUNCTION_BLOCK "FB_FillingTank"   // FB8, SCL
{ S7_Optimized_Access := 'FALSE' }
VERSION : 1.0
// MANTIS â€” Scene 3: Filling Tank
//  Fill and drain a tank using two discrete level sensors.
//  DB5: Instance DB for FB_FillingTank (non-optimized access)
// 
//  Factory I/O connections (ComDrvS7, Bool Inputs Offset=10):
//    Fill (high-level sensor)       â†’ %I10.0   TRUE = tank full
//    Discharge (low-level sensor)   â†’ %I10.1   TRUE = tank empty
//    FACTORY I/O (Running)          â†’ %I10.2   TRUE = simulation active
//    Fill valve                     â†’ %Q0.0
//    Filling (status indicator)     â†’ %Q0.1
//    Discharge valve                â†’ %Q0.2
//    Discharging (status indicator) â†’ %Q0.3
// 
//  DB5 byte layout (non-optimized, 18 bytes):
//    Byte 0   : SensorFill    (BOOL) â€” high-level: TRUE = tank full
//    Byte 2   : SensorDrain   (BOOL) â€” low-level:  TRUE = tank empty
//    Byte 4   : FIO_Running   (BOOL) â€” Factory I/O alive
//    Byte 6   : FillValve     (BOOL) â€” open fill valve
//    Byte 8   : Filling       (BOOL) â€” filling status indicator light
//    Byte 10  : DrainValve    (BOOL) â€” open drain valve
//    Byte 12  : Discharging   (BOOL) â€” discharging status indicator light
//    Byte 14  : IsFilling     (BOOL) â€” internal state: TRUE=filling, FALSE=draining
//    Byte 16  : Enable        (BOOL) â€” system enable (attack target)
//    Total = 18 bytes
// 
//  Normal cycle:
//    Start: tank empty (SensorDrain=TRUE) â†’ IsFilling=TRUE
//    Filling: FillValve=TRUE, Filling=TRUE â†’ tank rises
//    SensorFill=TRUE â†’ switch to drain: IsFilling=FALSE
//    Draining: DrainValve=TRUE, Discharging=TRUE â†’ tank empties
//    SensorDrain=TRUE â†’ switch to fill: IsFilling=TRUE â†’ repeat
// 
//  Attack surface:
//    Enable=FALSE     â†’ all valves close (DoS)
//    FillValve spoof  â†’ overflow or starvation
//    DrainValve spoof â†’ overflow or stuck full
   VAR
      SensorFill : Bool;   // byte 0.0 â€” Fill sensor (TRUE = tank full)
      _pad0 : Byte;   // byte 1
      SensorDrain : Bool;   // byte 2.0 â€” Discharge sensor (TRUE = tank empty)
      _pad1 : Byte;   // byte 3
      FIO_Running : Bool;   // byte 4.0 â€” Factory I/O alive
      _pad2 : Byte;   // byte 5
      FillValve : Bool;   // byte 6.0 â€” Fill valve actuator
      _pad3 : Byte;   // byte 7
      Filling : Bool;   // byte 8.0 â€” Filling indicator light
      _pad4 : Byte;   // byte 9
      DrainValve : Bool;   // byte 10.0 â€” Drain valve actuator
      _pad5 : Byte;   // byte 11
      Discharging : Bool;   // byte 12.0 â€” Discharging indicator light
      _pad6 : Byte;   // byte 13
      IsFilling : Bool := TRUE;   // byte 14.0 â€” State: TRUE=filling, FALSE=draining
      _pad7 : Byte;   // byte 15
      Enable : Bool := TRUE;   // byte 16.0 â€” System enable (attack target)
      _pad8 : Byte;   // byte 17 Total DB size: 18 bytes
   END_VAR
BEGIN
       IF NOT #FIO_Running OR NOT #Enable THEN
           // Safe state: close everything
           #FillValve := FALSE;
           #Filling := FALSE;
           #DrainValve := FALSE;
           #Discharging := FALSE;
       ELSIF #IsFilling THEN
           // Filling mode
           #FillValve := TRUE;
           #Filling := TRUE;
           #DrainValve := FALSE;
           #Discharging := FALSE;
           IF #SensorFill THEN
               #IsFilling := FALSE;    // Tank full â†’ switch to drain
           END_IF;
       ELSE
           // Draining mode
           #FillValve := FALSE;
           #Filling := FALSE;
           #DrainValve := TRUE;
           #Discharging := TRUE;
           IF #SensorDrain THEN
               #IsFilling := TRUE;     // Tank empty â†’ switch to fill
           END_IF;
       END_IF;
END_FUNCTION_BLOCK

FUNCTION_BLOCK "FB_FromAtoB"   // FB9, SCL
{ S7_Optimized_Access := 'FALSE' }
VERSION : 0.5
// MANTIS â€” Scene 1: From A to B
//  Transport a box on a conveyor until it reaches the sensor at the end.
//  DB3: Instance DB for FB_FromAtoB (non-optimized access)
// 
//  Factory I/O layout:
//    - Emitter automatically creates a box (not PLC-controlled)
//    - Conveyor moves the box from LEFT â†’ RIGHT  (%Q0.0)
//    - Sensor (diffuse) at the RIGHT end detects the box  (%I10.0)
// 
//  Driver config (Bool Inputs Offset=10, Bool Outputs Offset=0):
//    Sensor  â†’ %I10.0  (Factory I/O â†’ PLC)
//    Conveyor â†’ %Q0.0  (PLC â†’ Factory I/O)
// 
//  DB3 byte layout (non-optimized):
//    Byte 0   : Sensor   (BOOL)  â€” copied from %I10.0
//    Byte 1   : padding
//    Byte 2   : Conveyor (BOOL)  â€” copied to  %Q0.0
//    Byte 3   : padding
//    Byte 4   : Enable   (BOOL)  â€” system enable (default TRUE)
//    Byte 5   : padding
//    Total = 6 bytes
// 
//  Logic: Conveyor = Enable AND Sensor
//    Sensor True  â†’ path clear, no box â†’ Conveyor ON
//    Sensor False â†’ box detected        â†’ Conveyor OFF
//    Factory I/O reset clears all boxes â†’ sensor True â†’ conveyor starts.
// 
//  Vulnerability: Enable flag is read by logic but NEVER written by the FB.
//    An attacker who sets Enable=FALSE in DB3 stops the conveyor permanently.
   VAR
      Sensor : Bool;   // byte 0.0 â€” Sensor: box at end of conveyor
      _pad0 : Byte;   // byte 1 â€” padding
      Conveyor : Bool;   // byte 2.0 â€” Actuator: conveyor motor
      _pad1 : Byte;   // byte 3 â€” padding
      Enable : Bool := TRUE;   // byte 4.0 â€” System enable (default ON)
      _pad2 : Byte;   // byte 5 â€” padding
   END_VAR
BEGIN
       // Conveyor runs whenever enabled and no box at sensor
       #Conveyor := #Enable AND #Sensor;
END_FUNCTION_BLOCK

FUNCTION_BLOCK "FB_FromAtoB_SR"   // FB10, SCL
{ S7_Optimized_Access := 'FALSE' }
VERSION : 1.0
// MANTIS â€” Scene 2: From A to B (Set and Reset)
//  Transport a box from sensor A to sensor B using set/reset logic.
//  DB4: Instance DB for FB_FromAtoB_SR (non-optimized access)
// 
//  Factory I/O connections (ComDrvS7, Bool Inputs Offset=10):
//    Sensor A            â†’ %I10.0
//    Sensor B            â†’ %I10.1
//    FACTORY I/O Running â†’ %I10.2   (always TRUE while FIO is running)
//    Conveyor            â†’ %Q0.0
// 
//  DB4 byte layout (non-optimized, 12 bytes):
//    Byte 0   : SensorA     (BOOL)  â€” box at entry
//    Byte 1   : padding
//    Byte 2   : SensorB     (BOOL)  â€” box at exit
//    Byte 3   : padding
//    Byte 4   : FIO_Running (BOOL)  â€” Factory I/O alive signal
//    Byte 5   : padding
//    Byte 6   : Conveyor    (BOOL)  â€” conveyor motor output
//    Byte 7   : padding
//    Byte 8   : ConveyorRunning (BOOL) â€” SR latch state
//    Byte 9   : padding
//    Byte 10  : Enable      (BOOL)  â€” system enable (attack target)
//    Byte 11  : padding
//    Total = 12 bytes
// 
//  Normal cycle:
//    FIO starts  â†’ FIO_Running=TRUE, waiting for box
//    Box at A    â†’ SensorA=TRUE, SensorB=FALSE â†’ SET  conveyor ON
//    Box at B    â†’ SensorB=TRUE               â†’ RESET conveyor OFF
//    Auto-remover clears box â†’ SensorB=FALSE  â†’ next box triggers A
// 
//  Attack surface:
//    Enable=FALSE    â†’ full DoS (conveyor locked off)
//    SensorB spoof=TRUE  â†’ premature stop before box reaches exit
//    SensorB spoof=FALSE â†’ conveyor never stops (box overshoots)
   VAR
      SensorA : Bool;   // byte 0.0 â€” Sensor A: box at entry
      _pad0 : Byte;   // byte 1 â€” padding
      SensorB : Bool;   // byte 2.0 â€” Sensor B: box at exit
      _pad1 : Byte;   // byte 3 â€” padding
      FIO_Running : Bool;   // byte 4.0 â€” Factory I/O alive (always TRUE when running)
      _pad2 : Byte;   // byte 5 â€” padding
      Conveyor : Bool;   // byte 6.0 â€” Actuator: conveyor motor
      _pad3 : Byte;   // byte 7 â€” padding
      ConveyorRunning : Bool := FALSE;   // byte 8.0 â€” SR latch state
      _pad4 : Byte;   // byte 9 â€” padding
      Enable : Bool := TRUE;   // byte 10.0 â€” System enable (attack/DoS target)
      _pad5 : Byte;   // byte 11 â€” padding Total DB size: 12 bytes
   END_VAR
BEGIN
       // SR latch gated on FIO_Running
       //   FIO down            â†’ RESET (safe state: conveyor off)
       //   SensorB TRUE        â†’ RESET (box arrived at exit: stop)
       //   SensorA TRUE, B off â†’ SET   (box at entry, exit clear: start)
       //   otherwise           â†’ hold latch
       IF NOT #FIO_Running THEN
           #ConveyorRunning := FALSE;        // simulation not running â†’ stop
       ELSIF #SensorB THEN
           #ConveyorRunning := FALSE;        // RESET: box reached exit
       ELSIF #SensorA AND NOT #SensorB THEN
           #ConveyorRunning := TRUE;         // SET: box at entry, exit clear
       END_IF;

       // Gate final output on Enable (primary attack target)
       #Conveyor := #ConveyorRunning AND #Enable;
END_FUNCTION_BLOCK

FUNCTION_BLOCK "FB_LevelControl"   // FB11, SCL
{ S7_Optimized_Access := 'FALSE' }
VERSION : 0.4
// MANTIS â€” Scene 12: Level Control
//  Control the liquid level of a tank using fill/discharge valves.
//  DB21: Instance DB for FB_LevelControl (non-optimized access)
// 
//  Factory I/O layout:
//    - Tank with level meter, flow meter, fill valve, discharge valve
//    - Start/Stop/Reset buttons on control panel
//    - Start/Reset/Stop lights on panel
//    - SP and PV displays on panel
// 
//  Driver mapping (from Factory I/O):
//    SENSORS (Inputs):
//      NOTE: Use %I10.x (NOT %I0.x) because the PLC's
//      built-in physical DI module owns %IB0 and overwrites external writes.
//      Start        â†’ %I10.0  (BOOL)
//      Reset        â†’ %I10.1  (BOOL)
//      Stop         â†’ %I10.2  (BOOL)
//      FACTORY I/O (Running) â†’ %I10.3  (BOOL)
//      Level meter  â†’ %ID100  (REAL)  â€” tank level 0-10V
//      Flow meter   â†’ %ID104  (REAL)  â€” flow rate 0-10V
//      Setpoint     â†’ %ID108  (REAL)  â€” panel setpoint knob 0-10V
//        NOTE: Knob value is copied to SetpointIn ONLY while system is stopped.
//        Once Running=TRUE, SetpointIn freezes (OB_Main stops copying).
//        The PLC NEVER writes SetpointIn internally â€” it becomes a write-once
//        attack target. Use the knob to set the desired initial level before starting.
// 
//    ACTUATORS (Outputs):
//      Start light      â†’ %Q0.0   (BOOL)
//      Reset light      â†’ %Q0.1   (BOOL)
//      Stop light       â†’ %Q0.2   (BOOL)
//      Fill valve       â†’ %QD100  (REAL) â€” 0-10V
//      Discharge valve  â†’ %QD104  (REAL) â€” 0-10V
//      SP display       â†’ %QD108  (DINT) â€” setpoint display
//      PV display       â†’ %QD112  (DINT) â€” process value display
// 
//  DB21 byte layout (non-optimized):
//    Byte 0    : Start        (BOOL)   â€” %I10.0
//    Byte 1    : padding
//    Byte 2    : Reset        (BOOL)   â€” %I10.1
//    Byte 3    : padding
//    Byte 4    : Stop         (BOOL)   â€” %I10.2
//    Byte 5    : padding
//    Byte 6    : StartLight   (BOOL)   â€” %Q0.0
//    Byte 7    : padding
//    Byte 8    : ResetLight   (BOOL)   â€” %Q0.1
//    Byte 9    : padding
//    Byte 10   : StopLight    (BOOL)   â€” %Q0.2
//    Byte 11   : padding
//    Byte 12-15: LevelMeter   (REAL)   â€” %ID100
//    Byte 16-19: FlowMeter    (REAL)   â€” %ID104
//    Byte 20-23: SetpointIn   (REAL)   â€” from knob while stopped, frozen when running
//    Byte 24-27: FillValve    (REAL)   â€” %QD100
//    Byte 28-31: DischargeValve (REAL) â€” %QD104
//    Byte 32-35: SP_Display   (DINT)   â€” %QD108
//    Byte 36-39: PV_Display   (DINT)   â€” %QD112
//    Byte 40   : Running      (BOOL)   â€” internal: process running
//    Byte 41   : padding
//    Byte 42   : Enable       (BOOL)   â€” system enable (default TRUE)
//    Byte 43   : padding
//    Total = 44 bytes
// 
//  Normal operation:
//    Press Start â†’ Fill valve opens proportionally to error (simple P control)
//    Level meter reads â†’ PV display shows level
//    Setpoint knob â†’ SP display shows target
//    Fill valve adjusts to maintain level at setpoint
//    Press Stop â†’ Fill valve closes, discharge opens to drain
// 
//  Vulnerability 1: SetpointIn is used by controller but NEVER written by PLC logic.
//    OB_Main copies the Factory I/O knob to SetpointIn ONLY while Running=FALSE.
//    Once Running=TRUE, the copy stops and SetpointIn freezes at the knob value.
//    Attack: write any value to DB21 byte 20 while running.
//    SetpointIn=0.0 â†’ full drain. SetpointIn=5.0 â†’ 50% level.
//  Vulnerability 2: Enable flag is read by logic but NEVER written.
//    Setting Enable=FALSE stops fill valve and opens discharge.
//  Mapped to DB21 â€” order determines byte offsets (non-optimized)
   VAR
      Start : Bool;   // byte 0 â€” %I10.0 Start button
      _pad0 : Byte;   // byte 1
      Reset : Bool;   // byte 2 â€” %I10.1 Reset button
      _pad1 : Byte;   // byte 3
      Stop : Bool;   // byte 4 â€” %I10.2 Stop button
      _pad2 : Byte;   // byte 5
      StartLight : Bool;   // byte 6 â€” Start indicator
      _pad3 : Byte;   // byte 7
      ResetLight : Bool;   // byte 8 â€” Reset indicator
      _pad4 : Byte;   // byte 9
      StopLight : Bool;   // byte 10 â€” Stop indicator
      _pad5 : Byte;   // byte 11
      LevelMeter : Real;   // byte 12 â€” Tank level (0-10V)
      FlowMeter : Real;   // byte 16 â€” Flow rate (0-10V)
      SetpointIn : Real := 10.0;   // byte 20 â€” From knob (stopped) / frozen (running). WRITE-ONCE target.
      FillValve : Real;   // byte 24 â€” Fill valve opening (0-10V)
      DischargeValve : Real;   // byte 28 â€” Discharge valve opening (0-10V)
      SP_Display : DInt;   // byte 32 â€” SP display value
      PV_Display : DInt;   // byte 36 â€” PV display value
      Running : Bool := FALSE;   // byte 40 â€” Internal: process running
      _pad6 : Byte;   // byte 41
      Enable : Bool := TRUE;   // byte 42 â€” System enable (default ON)
      _pad7 : Byte;   // byte 43
   END_VAR
   VAR_TEMP
      error : Real;
      output : Real;
   END_VAR
BEGIN
       // â”€â”€ Safety gate: if Enable is FALSE, shut everything down â”€â”€
       IF NOT #Enable THEN
           #FillValve := 0.0;
           #DischargeValve := 10.0;     // Fully open discharge (0-10V range)
           #StartLight := FALSE;
           #StopLight := TRUE;
           #ResetLight := FALSE;
           #Running := FALSE;
           #SP_Display := 0;
           #PV_Display := REAL_TO_DINT(#LevelMeter);
           RETURN;
       END_IF;

       // â”€â”€ Update displays (scale 0-10V â†’ 0-100 for display) â”€â”€
       #SP_Display := REAL_TO_DINT(#SetpointIn * 10.0);
       #PV_Display := REAL_TO_DINT(#LevelMeter * 10.0);

       // â”€â”€ Button logic (matching Factory I/O convention) â”€â”€
       // Start: momentary â€” TRUE = pressed, FALSE = idle
       // Stop:  NC alternate â€” TRUE = not pressed (safe), FALSE = stop requested
       // Reset: momentary â€” TRUE = pressed, FALSE = idle
       IF #Start AND NOT #Running THEN
           #Running := TRUE;
       END_IF;

       IF NOT #Stop THEN
           #Running := FALSE;
       END_IF;

       // Auto-start: if Stop not pressed and Start not pressed, start automatically
       IF #Stop AND NOT #Start THEN
           #Running := TRUE;
       END_IF;

       IF #Reset THEN
           #Running := FALSE;
           #FillValve := 0.0;
           #DischargeValve := 0.0;
           #ResetLight := TRUE;
       ELSE
           #ResetLight := FALSE;
       END_IF;

       // â”€â”€ Indicator lights â”€â”€
       #StartLight := #Running;
       #StopLight := NOT #Running;

       // â”€â”€ Process control â”€â”€
       // Factory I/O tank valves use 0-10V range (NOT 0-100%)
       //   0V = fully closed, 10V = fully open
       IF #Running THEN
           // Simple proportional control
           #error := #SetpointIn - #LevelMeter;   // Both in 0-10V range

           IF #error > 0.0 THEN
               // Level below setpoint â†’ fill
               #output := #error * 1.0;          // P gain = 1.0 (0-10V range)
               IF #output > 10.0 THEN
                   #output := 10.0;
               END_IF;
               IF #output < 0.0 THEN
                   #output := 0.0;
               END_IF;
               #FillValve := #output;
               #DischargeValve := 0.0;
           ELSE
               // Level at or above setpoint â†’ stop filling, discharge excess
               #FillValve := 0.0;
               #output := - #error * 1.0;
               IF #output > 10.0 THEN
                   #output := 10.0;
               END_IF;
               IF #output < 0.0 THEN
                   #output := 0.0;
               END_IF;
               #DischargeValve := #output;
           END_IF;
       ELSE
           // Not running â†’ close everything
           #FillValve := 0.0;
           #DischargeValve := 0.0;
       END_IF;
END_FUNCTION_BLOCK

FUNCTION_BLOCK "FB_Palletizer"   // FB12, SCL
{ S7_Optimized_Access := 'FALSE' }
VERSION : 0.1
// MANTIS â€” Scene 13: Palletizer
//  Palletize cases in several layers.
//  DB22: I/O mapping
   VAR
      BoxAtEntry : Bool;   // 0.0
      _pad0 : Byte;
      BoxAtPickup : Bool;   // 2.0
      _pad1 : Byte;
      PalletReady : Bool;   // 4.0
      _pad2 : Byte;
      LayerComplete : Bool;   // 6.0
      _pad3 : Byte;
      ClampSensor : Bool;   // 8.0
      _pad4 : Byte;
      PosX : Real;   // 10
      PosZ : Real;   // 14
      ConveyorIn : Bool;   // 18.0
      _pad5 : Byte;
      Clamp : Bool;   // 20.0
      _pad6 : Byte;
      MoveX : Real;   // 22
      MoveZ : Real;   // 26
      ConveyorOut : Bool;   // 30.0
      _pad7 : Byte;
      Emitter : Bool;   // 32.0
      _pad8 : Byte;
      iState : Int := 0;
      BoxIndex : Int := 0;
      LayerIdx : Int := 0;
      BOXES_PER_LAYER : Int := 4;
      MAX_LAYERS : Int := 3;
      TOLERANCE : Real := 10.0;   // Placement positions (simplified grid)
      PlaceX : Real := 0.0;
      PlaceZ : Real := 0.0;
   END_VAR
BEGIN
       CASE #iState OF
           0: // Feed box
               #ConveyorIn := TRUE;
               #Emitter := TRUE;
               IF #BoxAtPickup THEN
                   #ConveyorIn := FALSE;
                   #Emitter := FALSE;
                   // Calculate placement position
                   #PlaceX := 200.0 + INT_TO_REAL(#BoxIndex MOD 2) * 200.0;
                   #PlaceZ := 100.0 + INT_TO_REAL(#LayerIdx) * 150.0;
                   #iState := 1;
               END_IF;

           1: // Move to pickup
               #MoveX := 0.0;  // Pickup X position
               #MoveZ := 0.0;  // Pickup Z (low)
               IF ABS(#PosX) < #TOLERANCE AND ABS(#PosZ) < #TOLERANCE THEN
                   #iState := 2;
               END_IF;

           2: // Clamp box
               #Clamp := TRUE;
               IF #ClampSensor THEN
                   #MoveZ := 200.0;  // Lift
                   #iState := 3;
               END_IF;

           3: // Move to place position
               IF ABS(#PosZ - 200.0) < #TOLERANCE THEN
                   #MoveX := #PlaceX;
                   #iState := 4;
               END_IF;

           4: // Lower to place
               IF ABS(#PosX - #PlaceX) < #TOLERANCE THEN
                   #MoveZ := #PlaceZ;
                   #iState := 5;
               END_IF;

           5: // Release
               IF ABS(#PosZ - #PlaceZ) < #TOLERANCE THEN
                   #Clamp := FALSE;
                   #BoxIndex := #BoxIndex + 1;
                   IF #BoxIndex >= #BOXES_PER_LAYER THEN
                       #BoxIndex := 0;
                       #LayerIdx := #LayerIdx + 1;
                       IF #LayerIdx >= #MAX_LAYERS THEN
                           #LayerIdx := 0;
                           #iState := 6;  // Pallet complete
                       ELSE
                           #iState := 0;
                       END_IF;
                   ELSE
                       #iState := 0;
                   END_IF;
               END_IF;

           6: // Output complete pallet
               #ConveyorOut := TRUE;
               IF NOT #PalletReady THEN
                   #ConveyorOut := FALSE;
                   #iState := 0;
               END_IF;
       END_CASE;
END_FUNCTION_BLOCK

FUNCTION_BLOCK "FB_PickPlaceBasic"   // FB13, SCL
{ S7_Optimized_Access := 'FALSE' }
VERSION : 0.1
// MANTIS â€” Scene 14: Pick & Place (Basic)
//  Pick and place items from one conveyor into another.
//  DB23: I/O mapping
   VAR
      ItemAtPick : Bool;   // 0.0
      _pad0 : Byte;
      ItemAtPlace : Bool;   // 2.0
      _pad1 : Byte;
      GripperClosed : Bool;   // 4.0
      _pad2 : Byte;
      ArmAtPick : Bool;   // 6.0
      _pad3 : Byte;
      ArmAtPlace : Bool;   // 8.0
      _pad4 : Byte;
      ConveyorIn : Bool;   // 10.0
      _pad5 : Byte;
      ConveyorOut : Bool;   // 12.0
      _pad6 : Byte;
      Gripper : Bool;   // 14.0
      _pad7 : Byte;
      ArmRotate : Bool;   // 16.0
      _pad8 : Byte;
      ArmUp : Bool;   // 18.0
      _pad9 : Byte;
      ArmDown : Bool;   // 20.0
      _pad10 : Byte;
      Emitter : Bool;   // 22.0
      _pad11 : Byte;
      iState : Int := 0;
   END_VAR
BEGIN
       #Emitter := TRUE;

       CASE #iState OF
           0: // Wait for item at pick position
               #ConveyorIn := TRUE;
               #ConveyorOut := TRUE;
               IF #ItemAtPick AND #ArmAtPick THEN
                   #ConveyorIn := FALSE;
                   #iState := 1;
               END_IF;

           1: // Lower arm
               #ArmDown := TRUE;
               #ArmUp := FALSE;
               IF NOT #ArmAtPick THEN  // Arm has moved down
                   #ArmDown := FALSE;
                   #iState := 2;
               END_IF;

           2: // Grip item
               #Gripper := TRUE;
               IF #GripperClosed THEN
                   #iState := 3;
               END_IF;

           3: // Raise arm
               #ArmUp := TRUE;
               #ArmDown := FALSE;
               IF #ArmAtPick THEN
                   #ArmUp := FALSE;
                   #iState := 4;
               END_IF;

           4: // Rotate to place
               #ArmRotate := TRUE;
               IF #ArmAtPlace THEN
                   #ArmRotate := FALSE;
                   #iState := 5;
               END_IF;

           5: // Lower arm
               #ArmDown := TRUE;
               IF NOT #ArmAtPlace THEN
                   #ArmDown := FALSE;
                   #iState := 6;
               END_IF;

           6: // Release
               #Gripper := FALSE;
               IF NOT #GripperClosed THEN
                   #ArmUp := TRUE;
                   #iState := 7;
               END_IF;

           7: // Return to pick position
               IF #ArmAtPlace THEN
                   #ArmUp := FALSE;
                   #ArmRotate := FALSE;  // Rotate back
                   #iState := 0;
               END_IF;
       END_CASE;
END_FUNCTION_BLOCK

FUNCTION_BLOCK "FB_PickPlaceXYZ"   // FB14, SCL
{ S7_Optimized_Access := 'FALSE' }
VERSION : 0.1
// MANTIS â€” Scene 15: Pick & Place XYZ
//  Place boxes onto pallets using a three-axis manipulator.
//  DB24: I/O mapping
   VAR
      BoxAtPick : Bool;   // 0.0
      _pad0 : Byte;
      PalletReady : Bool;   // 2.0
      _pad1 : Byte;
      GripperClosed : Bool;   // 4.0
      _pad2 : Byte;
      PosX : Real;   // 6
      PosY : Real;   // 10
      PosZ : Real;   // 14
      SetpointX : Real;   // 18
      SetpointY : Real;   // 22
      SetpointZ : Real;   // 26
      Gripper : Bool;   // 30.0
      _pad3 : Byte;
      ConveyorIn : Bool;   // 32.0
      _pad4 : Byte;
      ConveyorPallet : Bool;   // 34.0
      _pad5 : Byte;
      Emitter : Bool;   // 36.0
      _pad6 : Byte;
      iState : Int := 0;
      BoxIndex : Int := 0;
      TOLERANCE : Real := 10.0;   // Positions
      PICK_X : Real := 100.0;
      PICK_Y : Real := 100.0;
      PICK_Z : Real := 50.0;
      HOME_Z : Real := 300.0;
      PlaceX : Real := 0.0;
      PlaceY : Real := 0.0;
   END_VAR
BEGIN
       #Emitter := TRUE;

       CASE #iState OF
           0: // Wait for box
               #ConveyorIn := TRUE;
               #SetpointZ := #HOME_Z;
               IF #BoxAtPick THEN
                   #ConveyorIn := FALSE;
                   #iState := 1;
               END_IF;

           1: // Move to pick XY
               #SetpointX := #PICK_X;
               #SetpointY := #PICK_Y;
               IF ABS(#PosX - #PICK_X) < #TOLERANCE AND ABS(#PosY - #PICK_Y) < #TOLERANCE THEN
                   #iState := 2;
               END_IF;

           2: // Lower to pick
               #SetpointZ := #PICK_Z;
               IF ABS(#PosZ - #PICK_Z) < #TOLERANCE THEN
                   #Gripper := TRUE;
                   #iState := 3;
               END_IF;

           3: // Grip and raise
               IF #GripperClosed THEN
                   #SetpointZ := #HOME_Z;
                   #iState := 4;
               END_IF;

           4: // Move to place (grid pattern)
               IF ABS(#PosZ - #HOME_Z) < #TOLERANCE THEN
                   #PlaceX := 500.0 + INT_TO_REAL(#BoxIndex MOD 3) * 150.0;
                   #PlaceY := 100.0 + INT_TO_REAL(#BoxIndex / 3) * 150.0;
                   #SetpointX := #PlaceX;
                   #SetpointY := #PlaceY;
                   #iState := 5;
               END_IF;

           5: // Lower to place
               IF ABS(#PosX - #PlaceX) < #TOLERANCE AND ABS(#PosY - #PlaceY) < #TOLERANCE THEN
                   #SetpointZ := #PICK_Z;
                   #iState := 6;
               END_IF;

           6: // Release
               IF ABS(#PosZ - #PICK_Z) < #TOLERANCE THEN
                   #Gripper := FALSE;
                   #BoxIndex := #BoxIndex + 1;
                   IF #BoxIndex >= 9 THEN
                       #BoxIndex := 0;
                       #ConveyorPallet := TRUE;  // Eject full pallet
                   END_IF;
                   #SetpointZ := #HOME_Z;
                   #iState := 0;
               END_IF;
       END_CASE;
END_FUNCTION_BLOCK

FUNCTION_BLOCK "FB_ProductionLine"   // FB15, SCL
{ S7_Optimized_Access := 'FALSE' }
VERSION : 0.1
// MANTIS â€” Scene 16: Production Line
//  Produce matching lids and bases by controlling two machining centers.
//  DB25: I/O mapping
   VAR
      LidReady : Bool;   // 0.0
      _pad0 : Byte;
      BaseReady : Bool;   // 2.0
      _pad1 : Byte;
      LidAtAssembly : Bool;   // 4.0
      _pad2 : Byte;
      BaseAtAssembly : Bool;   // 6.0
      _pad3 : Byte;
      LidCount : Int;   // 8
      BaseCount : Int;   // 10
      LidMachine : Bool;   // 12.0
      _pad4 : Byte;
      BaseMachine : Bool;   // 14.0
      _pad5 : Byte;
      ConveyorLid : Bool;   // 16.0
      _pad6 : Byte;
      ConveyorBase : Bool;   // 18.0
      _pad7 : Byte;
      ConveyorOut : Bool;   // 20.0
      _pad8 : Byte;
      Emitter : Bool;   // 22.0
      _pad9 : Byte;
      LidsProduced : Int := 0;
      BasesProduced : Int := 0;
   END_VAR
BEGIN
       #Emitter := TRUE;
       #ConveyorOut := TRUE;

       // Run both machines to keep production balanced
       // Simple balancing: if one is ahead, slow it down
       IF #LidsProduced <= #BasesProduced THEN
           #LidMachine := TRUE;
       ELSE
           #LidMachine := FALSE;  // Pause lid production to balance
       END_IF;

       IF #BasesProduced <= #LidsProduced THEN
           #BaseMachine := TRUE;
       ELSE
           #BaseMachine := FALSE;
       END_IF;

       // Count produced items
       IF #LidReady THEN
           #ConveyorLid := TRUE;
           #LidsProduced := #LidsProduced + 1;
           #LidCount := #LidsProduced;
       END_IF;

       IF #BaseReady THEN
           #ConveyorBase := TRUE;
           #BasesProduced := #BasesProduced + 1;
           #BaseCount := #BasesProduced;
       END_IF;

       // Enable output when both parts are at assembly
       IF #LidAtAssembly AND #BaseAtAssembly THEN
           #ConveyorOut := TRUE;
       END_IF;
END_FUNCTION_BLOCK

FUNCTION_BLOCK "FB_QueueItems"   // FB16, SCL
{ S7_Optimized_Access := 'FALSE' }
VERSION : 0.1
// MANTIS â€” Scene 4: Queue of Items (Counters)
//  Load and unload three boxes onto a conveyor using counters.
//  DB13: I/O mapping
   VAR
      AtEntry : Bool;   // 0.0
      _pad0 : Byte;
      AtExit : Bool;   // 2.0
      _pad1 : Byte;
      Conveyor : Bool;   // 4.0
      _pad2 : Byte;
      Emitter : Bool;   // 6.0
      _pad3 : Byte;
      Remover : Bool;   // 8.0
      _pad4 : Byte;
      BoxCounter : Int;   // 10
      iState : Int := 0;
      BoxCount : Int := 0;
      TARGET_COUNT : Int := 3;
      PrevAtEntry : Bool := FALSE;
   END_VAR
BEGIN
       CASE #iState OF
           0: // Loading phase â€” emit boxes until count reached
               #Conveyor := TRUE;
               #Remover := FALSE;

               IF #BoxCount < #TARGET_COUNT THEN
                   #Emitter := TRUE;
                   // Count on rising edge of AtEntry
                   IF #AtEntry AND NOT #PrevAtEntry THEN
                       #BoxCount := #BoxCount + 1;
                   END_IF;
               ELSE
                   #Emitter := FALSE;
                   #iState := 1;
               END_IF;

           1: // Unloading phase â€” remove all boxes
               #Conveyor := TRUE;
               #Remover := TRUE;
               #Emitter := FALSE;

               IF #AtExit THEN
                   #BoxCount := #BoxCount - 1;
                   IF #BoxCount <= 0 THEN
                       #BoxCount := 0;
                       #iState := 0;
                   END_IF;
               END_IF;
       END_CASE;

       #PrevAtEntry := #AtEntry;
       #BoxCounter := #BoxCount;
END_FUNCTION_BLOCK

FUNCTION_BLOCK "FB_SeparatingStation"   // FB17, SCL
{ S7_Optimized_Access := 'FALSE' }
VERSION : 0.1
// MANTIS â€” Scene 17: Separating Station
//  Separate blue and green parts into two conveyors.
//  DB26: I/O mapping
   VAR
      PartAtEntry : Bool;   // 0.0
      _pad0 : Byte;
      VisionSensor : Int;   // 2 (0=none, 1=green, 2=blue)
      AtDiverter : Bool;   // 4.0
      _pad1 : Byte;
      AtExitLeft : Bool;   // 6.0
      _pad2 : Byte;
      AtExitRight : Bool;   // 8.0
      _pad3 : Byte;
      ConveyorIn : Bool;   // 10.0
      _pad4 : Byte;
      ConveyorLeft : Bool;   // 12.0
      _pad5 : Byte;
      ConveyorRight : Bool;   // 14.0
      _pad6 : Byte;
      Diverter : Bool;   // 16.0 (FALSE=left/green, TRUE=right/blue)
      _pad7 : Byte;
      Emitter : Bool;   // 18.0
      _pad8 : Byte;
      RemoverLeft : Bool;   // 20.0
      _pad9 : Byte;
      RemoverRight : Bool;   // 22.0
      _pad10 : Byte;
      DetectedColor : Int := 0;
   END_VAR
BEGIN
       #Emitter := TRUE;
       #ConveyorIn := TRUE;
       #ConveyorLeft := TRUE;
       #ConveyorRight := TRUE;
       #RemoverLeft := TRUE;
       #RemoverRight := TRUE;

       // Detect color when part enters
       IF #PartAtEntry AND #VisionSensor > 0 THEN
           #DetectedColor := #VisionSensor;
       END_IF;

       // Set diverter based on detected color
       IF #AtDiverter THEN
           IF #DetectedColor = 1 THEN
               #Diverter := FALSE;  // Green -> left
           ELSIF #DetectedColor = 2 THEN
               #Diverter := TRUE;   // Blue -> right
           END_IF;
       END_IF;
END_FUNCTION_BLOCK

